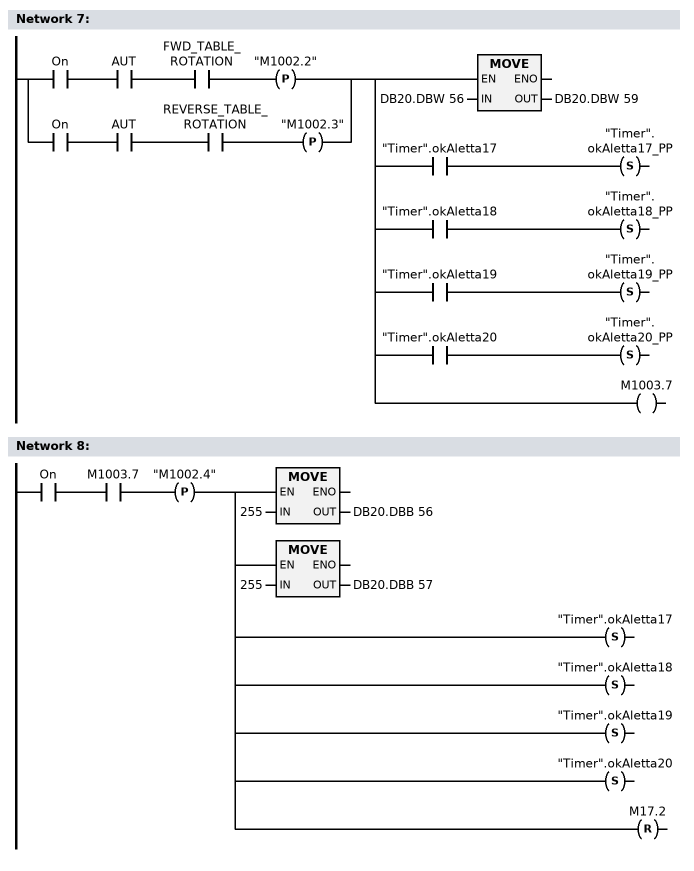
[picture p85: FC53 - REWORK networks 7-8]
NETWORK
TITLE =
      A     "On";
      A     "AUT";
      A     "FWD_TABLE_ROTATION";
      FP    "M1002.2";
      O(;
      A     "On";
      A     "AUT";
      A     "REVERSE_TABLE_ROTATION";
      FP    "M1002.3";
      );
      =     L 0.0;
      A     L 0.0;
      JNB   _009;
      L     DB20.DBW 56;
      T     DB20.DBW 59;
_009: NOP   0;
      A     L 0.0;
      A     "Timer".okAletta17;
      S     "Timer".okAletta17_PP;
      A     L 0.0;
      A     "Timer".okAletta18;
      S     "Timer".okAletta18_PP;
      A     L 0.0;
      A     "Timer".okAletta19;
      S     "Timer".okAletta19_PP;
      A     L 0.0;
      A     "Timer".okAletta20;
      S     "Timer".okAletta20_PP;
      A     L 0.0;
      BLD   102;
      =     "M1003.7";
NETWORK
TITLE =
      A     "On";
      A     "M1003.7";
      FP    "M1002.4";
      =     L 0.0;
      A     L 0.0;
      JNB   _00a;
      L     255;
      T     DB20.DBB 56;
_00a: NOP   0;
      A     L 0.0;
      JNB   _00b;
      L     255;
      T     DB20.DBB 57;
_00b: NOP   0;
      A     L 0.0;
      BLD   102;
      S     "Timer".okAletta17;
      A     L 0.0;
      BLD   102;
      S     "Timer".okAletta18;
      A     L 0.0;
      BLD   102;
      S     "Timer".okAletta19;
      A     L 0.0;
      BLD   102;
      S     "Timer".okAletta20;
      A     L 0.0;
      BLD   102;
      R     "M17.2";
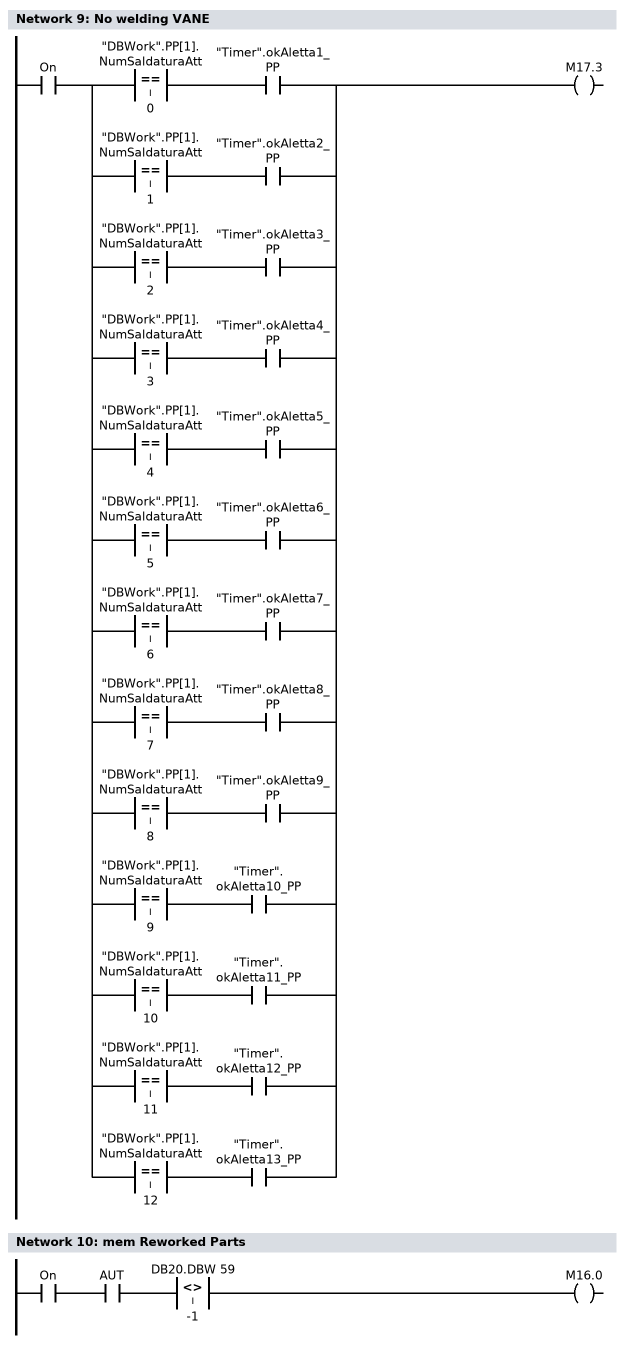
NETWORK
TITLE = No welding VANE
      A     "On";
      A(;
      A(;
      L     "DBWork".PP[1].NumSaldaturaAtt;
      L     0;
      ==I;
      );
      A     "Timer".okAletta1_PP;
      O;
      A(;
      L     "DBWork".PP[1].NumSaldaturaAtt;
      L     1;
      ==I;
      );
      A     "Timer".okAletta2_PP;
      O;
      A(;
      L     "DBWork".PP[1].NumSaldaturaAtt;
      L     2;
      ==I;
      );
      A     "Timer".okAletta3_PP;
      O;
      A(;
      L     "DBWork".PP[1].NumSaldaturaAtt;
      L     3;
      ==I;
      );
      A     "Timer".okAletta4_PP;
      O;
      A(;
      L     "DBWork".PP[1].NumSaldaturaAtt;
      L     4;
      ==I;
      );
      A     "Timer".okAletta5_PP;
      O;
      A(;
      L     "DBWork".PP[1].NumSaldaturaAtt;
      L     5;
      ==I;
      );
      A     "Timer".okAletta6_PP;
      O;
      A(;
      L     "DBWork".PP[1].NumSaldaturaAtt;
      L     6;
      ==I;
      );
      A     "Timer".okAletta7_PP;
      O;
      A(;
      L     "DBWork".PP[1].NumSaldaturaAtt;
      L     7;
      ==I;
      );
      A     "Timer".okAletta8_PP;
      O;
      A(;
      L     "DBWork".PP[1].NumSaldaturaAtt;
      L     8;
      ==I;
      );
      A     "Timer".okAletta9_PP;
      O;
      A(;
      L     "DBWork".PP[1].NumSaldaturaAtt;
      L     9;
      ==I;
      );
      A     "Timer".okAletta10_PP;
      O;
      A(;
      L     "DBWork".PP[1].NumSaldaturaAtt;
      L     10;
      ==I;
      );
      A     "Timer".okAletta11_PP;
      O;
      A(;
      L     "DBWork".PP[1].NumSaldaturaAtt;
      L     11;
      ==I;
      );
      A     "Timer".okAletta12_PP;
      O;
      A(;
      L     "DBWork".PP[1].NumSaldaturaAtt;
      L     12;
      ==I;
      );
      A     "Timer".okAletta13_PP;
      );
      =     "M17.3";
NETWORK
TITLE = mem Reworked Parts
      A     "On";
      A     "AUT";
      A(;
      L     DB20.DBW 59;
      L     -1;
      <>I;
      );
      =     "M16.0";
END_FUNCTION

FUNCTION "FC81 - GEST AXIS" : VOID	// FC 81
VERSION : 0.1
VAR_TEMP
  AttualPos : DINT ;
  AttualPosR : REAL ;
  Override : INT ;
  AuxRelative : DINT ;
  JogRelative : BOOL ;
END_VAR
BEGIN
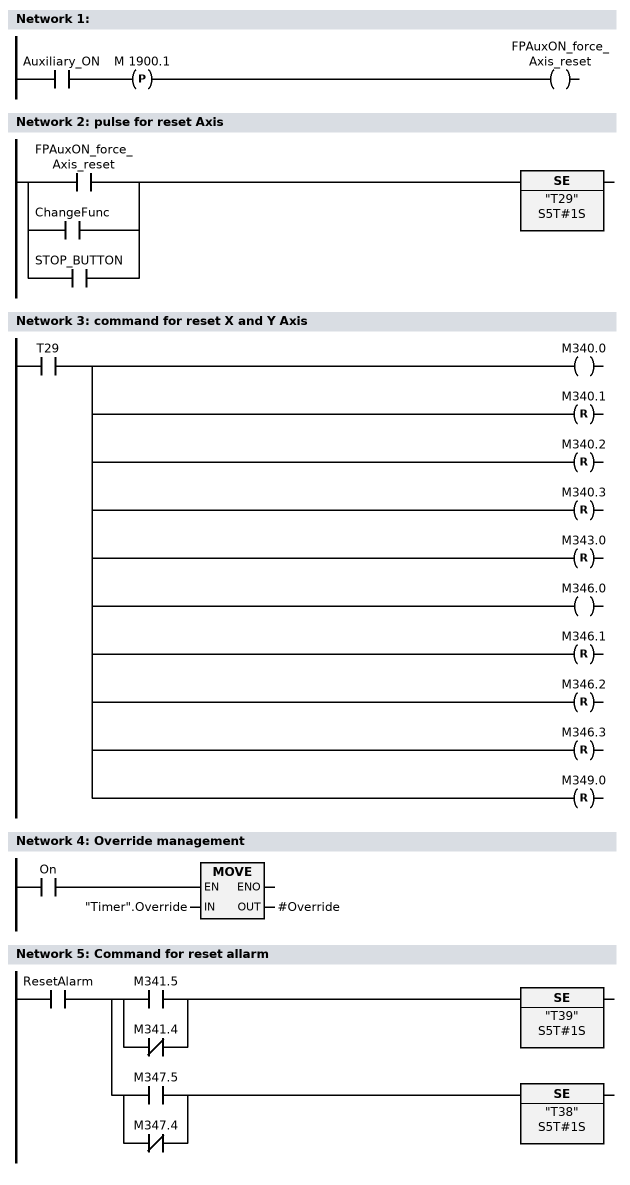
NETWORK
TITLE =
      A     "Auxiliary_ON";
      FP    M 1900.1;
      =     "FPAuxON_force_Axis_reset";
NETWORK
TITLE = pulse for reset Axis
      O     "FPAuxON_force_Axis_reset";
      O     "ChangeFunc";
      O     "STOP_BUTTON";
      L     S5T#1S;
      SE    "T29";
NETWORK
TITLE = command for reset X and Y Axis
      A     "T29";
      =     "M340.0";
      R     "M340.1";
      R     "M340.2";
      R     "M340.3";
      R     "M343.0";
      =     "M346.0";
      R     "M346.1";
      R     "M346.2";
      R     "M346.3";
      R     "M349.0";
NETWORK
TITLE = Override management
//"DatiMacchina".AcesXYZC_Override_Aux
      A     "On";
      JNB   _001;
      L     "Timer".Override;
      T     #Override;
_001: NOP   0;
NETWORK
TITLE = Command for reset allarm
      A     "ResetAlarm";
      =     L 15.0;
      A     L 15.0;
      A(;
      O     "M341.5";
      ON    "M341.4";
      );
      L     S5T#1S;
      SE    "T39";
      A     L 15.0;
      A(;
      O     "M347.5";
      ON    "M347.4";
      );
      L     S5T#1S;
      SE    "T38";
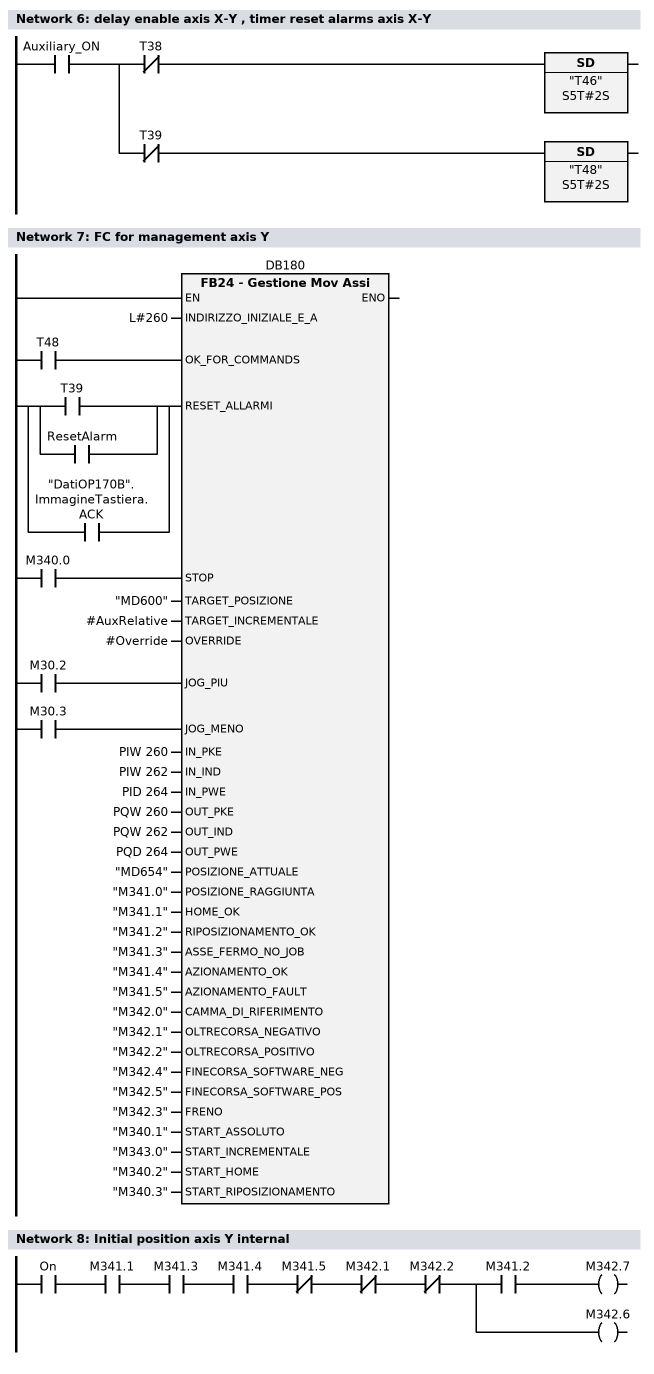
NETWORK
TITLE = delay enable axis X-Y , timer reset alarms axis X-Y
      A     "Auxiliary_ON";
      =     L 15.0;
      A     L 15.0;
      AN    "T38";
      L     S5T#2S;
      SD    "T46";
      A     L 15.0;
      AN    "T39";
      L     S5T#2S;
      SD    "T48";
NETWORK
TITLE = FC for management axis Y
      A     "T48";
      =     L 15.0;
      BLD   103;
      A(;
      O     "T39";
      O     "ResetAlarm";
      O     "DatiOP170B".ImmagineTastiera.ACK;
      );
      =     L 15.1;
      BLD   103;
      A     "M340.0";
      =     L 15.2;
      BLD   103;
      A     "M30.2";
      =     L 15.3;
      BLD   103;
      A     "M30.3";
      =     L 15.4;
      BLD   103;
      CALL  "FB24 - Gestione Mov Assi" , "DB180" (
           INDIRIZZO_INIZIALE_E_A   := L#260,
           OK_FOR_COMMANDS          := L 15.0,
           RESET_ALLARMI            := L 15.1,
           STOP                     := L 15.2,
           TARGET_POSIZIONE         := "MD600",
           TARGET_INCREMENTALE      := #AuxRelative,
           OVERRIDE                 := #Override,
           JOG_PIU                  := L 15.3,
           JOG_MENO                 := L 15.4,
           IN_PKE                   := PIW 260,
           IN_IND                   := PIW 262,
           IN_PWE                   := PID 264,
           OUT_PKE                  := PQW 260,
           OUT_IND                  := PQW 262,
           OUT_PWE                  := PQD 264,
           POSIZIONE_ATTUALE        := "MD654",
           POSIZIONE_RAGGIUNTA      := "M341.0",
           HOME_OK                  := "M341.1",
           RIPOSIZIONAMENTO_OK      := "M341.2",
           ASSE_FERMO_NO_JOB        := "M341.3",
           AZIONAMENTO_OK           := "M341.4",
           AZIONAMENTO_FAULT        := "M341.5",
           CAMMA_DI_RIFERIMENTO     := "M342.0",
           OLTRECORSA_NEGATIVO      := "M342.1",
           OLTRECORSA_POSITIVO      := "M342.2",
           FINECORSA_SOFTWARE_NEG   := "M342.4",
           FINECORSA_SOFTWARE_POS   := "M342.5",
           FRENO                    := "M342.3",
           START_ASSOLUTO           := "M340.1",
           START_INCREMENTALE       := "M343.0",
           START_HOME               := "M340.2",
           START_RIPOSIZIONAMENTO   := "M340.3");
      NOP   0;
NETWORK
TITLE = Initial position axis Y internal
      A     "On";
      A     "M341.1";
      A     "M341.3";
      A     "M341.4";
      AN    "M341.5";
      AN    "M342.1";
      AN    "M342.2";
      =     L 15.0;
      A     L 15.0;
      A     "M341.2";
      =     "M342.7";
      A     L 15.0;
      BLD   102;
      =     "M342.6";
NETWORK
TITLE = Axis X Management
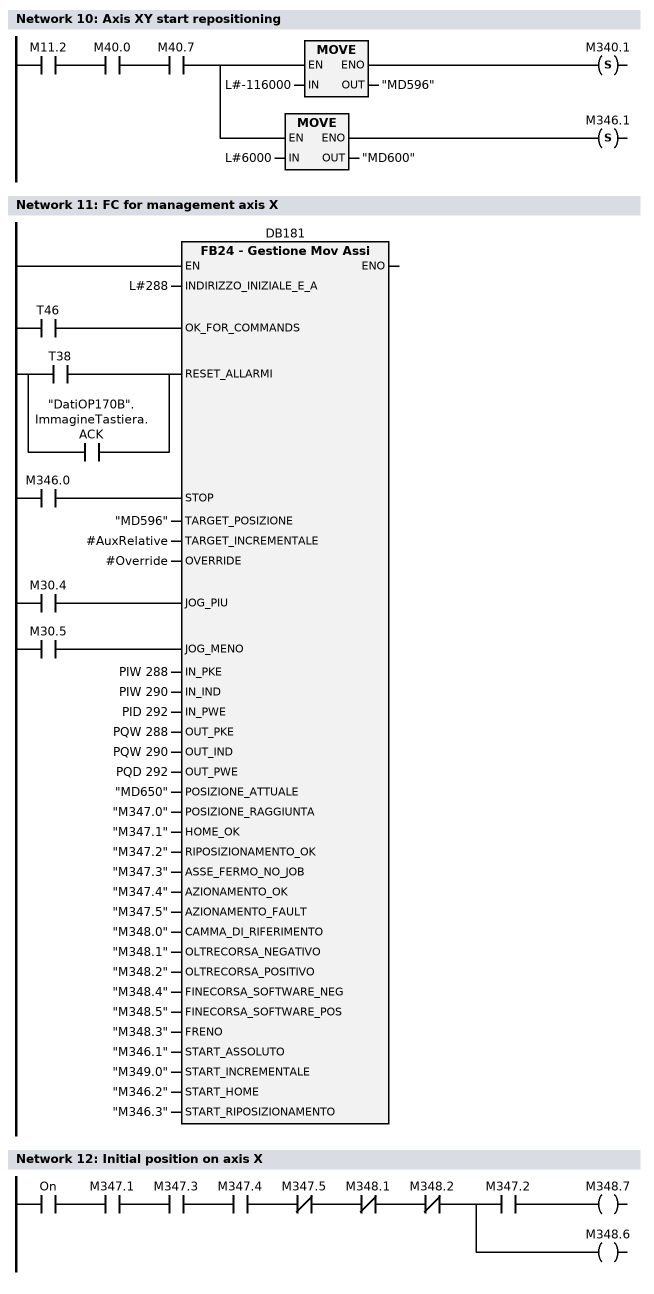
NETWORK
TITLE = Axis XY start repositioning
      A     "M11.2";
      A     "M40.0";
      A     "M40.7";
      =     L 15.0;
      A     L 15.0;
      JNB   _002;
      L     L#-116000;
      T     "MD596";
      SET;
      SAVE;
      CLR;
_002: A     BR;
      S     "M340.1";
      A     L 15.0;
      JNB   _003;
      L     L#6000;
      T     "MD600";
      SET;
      SAVE;
      CLR;
_003: A     BR;
      S     "M346.1";
NETWORK
TITLE = FC for management axis X
      A     "T46";
      =     L 15.0;
      BLD   103;
      A(;
      O     "T38";
      O     "DatiOP170B".ImmagineTastiera.ACK;
      );
      =     L 15.1;
      BLD   103;
      A     "M346.0";
      =     L 15.2;
      BLD   103;
      A     "M30.4";
      =     L 15.3;
      BLD   103;
      A     "M30.5";
      =     L 15.4;
      BLD   103;
      CALL  "FB24 - Gestione Mov Assi" , "DB181" (
           INDIRIZZO_INIZIALE_E_A   := L#288,
           OK_FOR_COMMANDS          := L 15.0,
           RESET_ALLARMI            := L 15.1,
           STOP                     := L 15.2,
           TARGET_POSIZIONE         := "MD596",
           TARGET_INCREMENTALE      := #AuxRelative,
           OVERRIDE                 := #Override,
           JOG_PIU                  := L 15.3,
           JOG_MENO                 := L 15.4,
           IN_PKE                   := PIW 288,
           IN_IND                   := PIW 290,
           IN_PWE                   := PID 292,
           OUT_PKE                  := PQW 288,
           OUT_IND                  := PQW 290,
           OUT_PWE                  := PQD 292,
           POSIZIONE_ATTUALE        := "MD650",
           POSIZIONE_RAGGIUNTA      := "M347.0",
           HOME_OK                  := "M347.1",
           RIPOSIZIONAMENTO_OK      := "M347.2",
           ASSE_FERMO_NO_JOB        := "M347.3",
           AZIONAMENTO_OK           := "M347.4",
           AZIONAMENTO_FAULT        := "M347.5",
           CAMMA_DI_RIFERIMENTO     := "M348.0",
           OLTRECORSA_NEGATIVO      := "M348.1",
           OLTRECORSA_POSITIVO      := "M348.2",
           FINECORSA_SOFTWARE_NEG   := "M348.4",
           FINECORSA_SOFTWARE_POS   := "M348.5",
           FRENO                    := "M348.3",
           START_ASSOLUTO           := "M346.1",
           START_INCREMENTALE       := "M349.0",
           START_HOME               := "M346.2",
           START_RIPOSIZIONAMENTO   := "M346.3");
      NOP   0;
NETWORK
TITLE = Initial position on axis X
      A     "On";
      A     "M347.1";
      A     "M347.3";
      A     "M347.4";
      AN    "M347.5";
      AN    "M348.1";
      AN    "M348.2";
      =     L 15.0;
      A     L 15.0;
      A     "M347.2";
      =     "M348.7";
      A     L 15.0;
      BLD   102;
      =     "M348.6";
END_FUNCTION

FUNCTION "FC117 - ERROR TOOL" : VOID	// FC 117
VERSION : 0.1
BEGIN
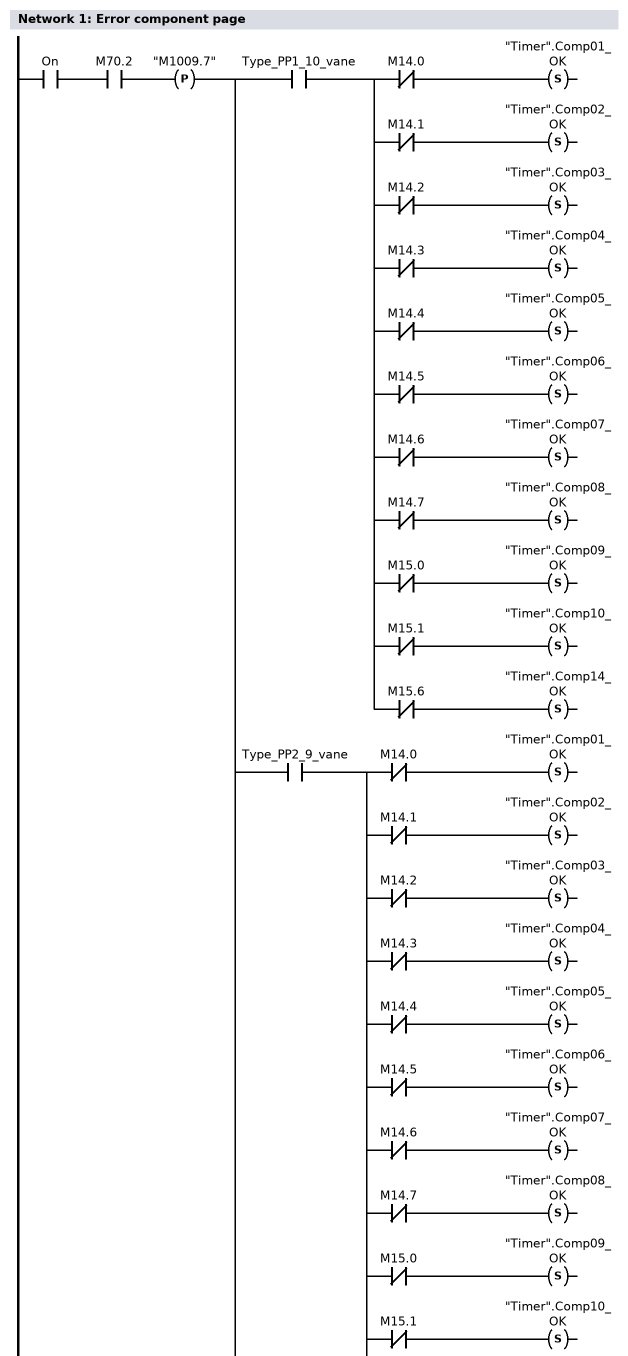
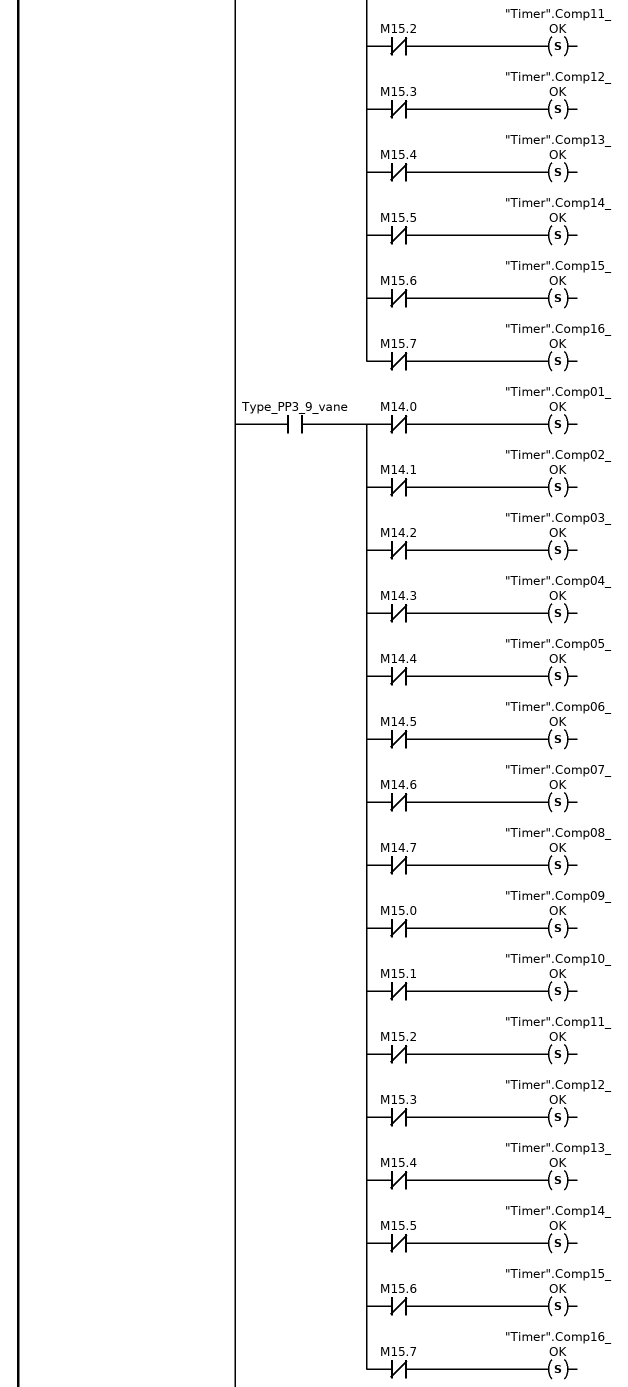
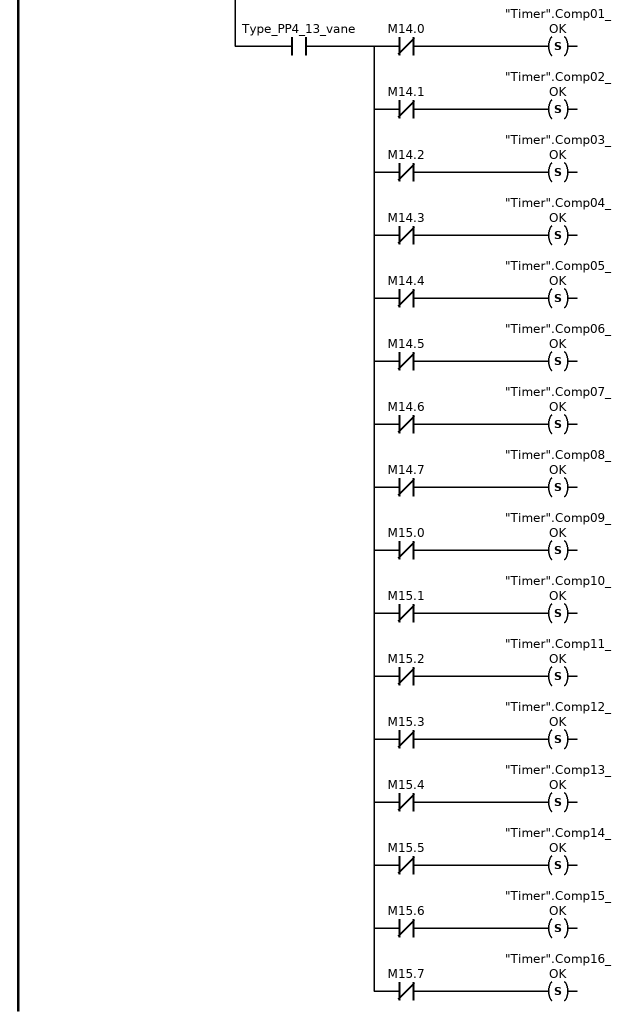
NETWORK
TITLE = Error component page
      A     "On";
      A     "M70.2";
      FP    "M1009.7";
      =     L 0.0;
      A     L 0.0;
      A     "Type_PP1_10_vane";
      =     L 0.1;
      A     L 0.1;
      AN    "M14.0";
      S     "Timer".Comp01_OK;
      A     L 0.1;
      AN    "M14.1";
      S     "Timer".Comp02_OK;
      A     L 0.1;
      AN    "M14.2";
      S     "Timer".Comp03_OK;
      A     L 0.1;
      AN    "M14.3";
      S     "Timer".Comp04_OK;
      A     L 0.1;
      AN    "M14.4";
      S     "Timer".Comp05_OK;
      A     L 0.1;
      AN    "M14.5";
      S     "Timer".Comp06_OK;
      A     L 0.1;
      AN    "M14.6";
      S     "Timer".Comp07_OK;
      A     L 0.1;
      AN    "M14.7";
      S     "Timer".Comp08_OK;
      A     L 0.1;
      AN    "M15.0";
      S     "Timer".Comp09_OK;
      A     L 0.1;
      AN    "M15.1";
      S     "Timer".Comp10_OK;
      A     L 0.1;
      AN    "M15.6";
      S     "Timer".Comp14_OK;
      A     L 0.0;
      A     "Type_PP2_9_vane";
      =     L 0.1;
      A     L 0.1;
      AN    "M14.0";
      S     "Timer".Comp01_OK;
      A     L 0.1;
      AN    "M14.1";
      S     "Timer".Comp02_OK;
      A     L 0.1;
      AN    "M14.2";
      S     "Timer".Comp03_OK;
      A     L 0.1;
      AN    "M14.3";
      S     "Timer".Comp04_OK;
      A     L 0.1;
      AN    "M14.4";
      S     "Timer".Comp05_OK;
      A     L 0.1;
      AN    "M14.5";
      S     "Timer".Comp06_OK;
      A     L 0.1;
      AN    "M14.6";
      S     "Timer".Comp07_OK;
      A     L 0.1;
      AN    "M14.7";
      S     "Timer".Comp08_OK;
      A     L 0.1;
      AN    "M15.0";
      S     "Timer".Comp09_OK;
      A     L 0.1;
      AN    "M15.1";
      S     "Timer".Comp10_OK;
      A     L 0.1;
      AN    "M15.2";
      S     "Timer".Comp11_OK;
      A     L 0.1;
      AN    "M15.3";
      S     "Timer".Comp12_OK;
      A     L 0.1;
      AN    "M15.4";
      S     "Timer".Comp13_OK;
      A     L 0.1;
      AN    "M15.5";
      S     "Timer".Comp14_OK;
      A     L 0.1;
      AN    "M15.6";
      S     "Timer".Comp15_OK;
      A     L 0.1;
      AN    "M15.7";
      S     "Timer".Comp16_OK;
      A     L 0.0;
      A     "Type_PP3_9_vane";
      =     L 0.1;
      A     L 0.1;
      AN    "M14.0";
      S     "Timer".Comp01_OK;
      A     L 0.1;
      AN    "M14.1";
      S     "Timer".Comp02_OK;
      A     L 0.1;
      AN    "M14.2";
      S     "Timer".Comp03_OK;
      A     L 0.1;
      AN    "M14.3";
      S     "Timer".Comp04_OK;
      A     L 0.1;
      AN    "M14.4";
      S     "Timer".Comp05_OK;
      A     L 0.1;
      AN    "M14.5";
      S     "Timer".Comp06_OK;
      A     L 0.1;
      AN    "M14.6";
      S     "Timer".Comp07_OK;
      A     L 0.1;
      AN    "M14.7";
      S     "Timer".Comp08_OK;
      A     L 0.1;
      AN    "M15.0";
      S     "Timer".Comp09_OK;
      A     L 0.1;
      AN    "M15.1";
      S     "Timer".Comp10_OK;
      A     L 0.1;
      AN    "M15.2";
      S     "Timer".Comp11_OK;
      A     L 0.1;
      AN    "M15.3";
      S     "Timer".Comp12_OK;
      A     L 0.1;
      AN    "M15.4";
      S     "Timer".Comp13_OK;
      A     L 0.1;
      AN    "M15.5";
      S     "Timer".Comp14_OK;
      A     L 0.1;
      AN    "M15.6";
      S     "Timer".Comp15_OK;
      A     L 0.1;
      AN    "M15.7";
      S     "Timer".Comp16_OK;
      A     L 0.0;
      A     "Type_PP4_13_vane";
      =     L 0.1;
      A     L 0.1;
      AN    "M14.0";
      S     "Timer".Comp01_OK;
      A     L 0.1;
      AN    "M14.1";
      S     "Timer".Comp02_OK;
      A     L 0.1;
      AN    "M14.2";
      S     "Timer".Comp03_OK;
      A     L 0.1;
      AN    "M14.3";
      S     "Timer".Comp04_OK;
      A     L 0.1;
      AN    "M14.4";
      S     "Timer".Comp05_OK;
      A     L 0.1;
      AN    "M14.5";
      S     "Timer".Comp06_OK;
      A     L 0.1;
      AN    "M14.6";
      S     "Timer".Comp07_OK;
      A     L 0.1;
      AN    "M14.7";
      S     "Timer".Comp08_OK;
      A     L 0.1;
      AN    "M15.0";
      S     "Timer".Comp09_OK;
      A     L 0.1;
      AN    "M15.1";
      S     "Timer".Comp10_OK;
      A     L 0.1;
      AN    "M15.2";
      S     "Timer".Comp11_OK;
      A     L 0.1;
      AN    "M15.3";
      S     "Timer".Comp12_OK;
      A     L 0.1;
      AN    "M15.4";
      S     "Timer".Comp13_OK;
      A     L 0.1;
      AN    "M15.5";
      S     "Timer".Comp14_OK;
      A     L 0.1;
      AN    "M15.6";
      S     "Timer".Comp15_OK;
      A     L 0.1;
      AN    "M15.7";
      S     "Timer".Comp16_OK;
END_FUNCTION

FUNCTION "TimeOut" : VOID	// FC 800
TITLE = Gestione timeout movimento
FAMILY : GCLib
NAME : TimeOut
VERSION : 1.0
VAR_INPUT
  Condizione1 : BOOL ;
  Condizione2 : BOOL ;
  Contatore : COUNTER ;
  Reset : BOOL ;
  Tempo_TimeOut : INT ;
END_VAR
VAR_IN_OUT
  TimeOut_Condizione1 : BOOL ;
  TimeOut_Condizione2 : BOOL ;
END_VAR
BEGIN
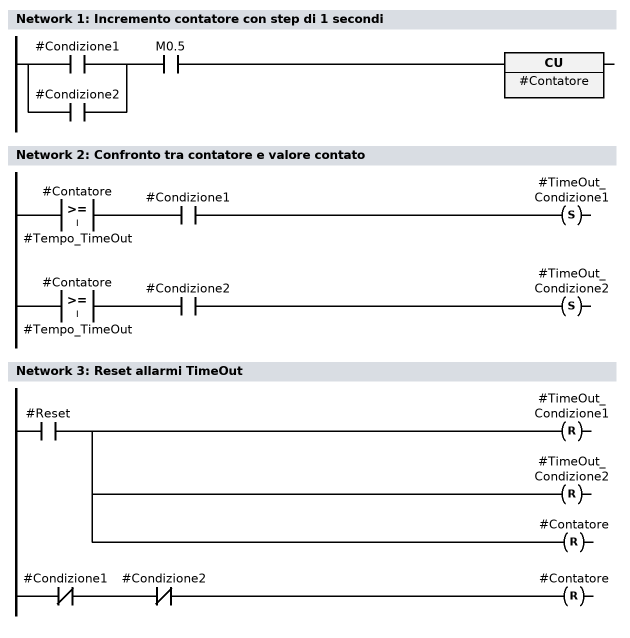
NETWORK
TITLE = Incremento contatore con step di 1 secondi
      A     #Condizione1;
      O     #Condizione2;
      A     "M0.5";
      CU    #Contatore;
NETWORK
TITLE = Confronto tra contatore e valore contato
      L     #Contatore;
      L     #Tempo_TimeOut;
      >=I;
      A     #Condizione1;
      S     #TimeOut_Condizione1;
      L     #Contatore;
      L     #Tempo_TimeOut;
      >=I;
      A     #Condizione2;
      S     #TimeOut_Condizione2;
NETWORK
TITLE = Reset allarmi TimeOut
      A     #Reset;
      R     #TimeOut_Condizione1;
      R     #TimeOut_Condizione2;
      R     #Contatore;
      AN    #Condizione1;
      AN    #Condizione2;
      R     #Contatore;
END_FUNCTION

DATA_BLOCK "DI_Balluff1"	// DB 5
VERSION : 0.0
"BALLUFF"
BEGIN
END_DATA_BLOCK

DATA_BLOCK "DatiOP170B"	// DB 7
TITLE = Dati interfaccia tra PLC e OP170B
FAMILY : GCLib
VERSION : 0.1
  STRUCT
   NumeroPagina : STRUCT
    TipoPaginaCorrente : WORD ;
    NumeroPaginaCorrente : INT ;
    Riservato1 : WORD ;
    Riservato2 : WORD ;
    Riservato3 : WORD ;
   END_STRUCT ;
   BufferOrdini : STRUCT
    NU : BYTE ;
    NumeroOrdine : BYTE ;
    Parametro1 : WORD ;
    Parametro2 : WORD ;
    Parametro3 : WORD ;
   END_STRUCT ;
   Coordinazione : STRUCT
    NU : BYTE ;
    BitAvvio : BOOL ;
    TipoFunzionamento : BOOL ;
    BitAttivita : BOOL ;
    Riservato1 : BOOL ;
    Riservato2 : BOOL ;
    Riservato3 : BOOL ;
    Riservato4 : BOOL ;
    Riservato5 : BOOL ;
    Riservata : WORD ;
   END_STRUCT ;
   ImmagineLED : STRUCT
    Bit0_F1 : BOOL ;
    Bit1_F1 : BOOL ;
    Bit0_F2 : BOOL ;
    Bit1_F2 : BOOL ;
    Bit0_F3 : BOOL ;
    Bit1_F3 : BOOL ;
    Bit0_F4 : BOOL ;
    Bit1_F4 : BOOL ;
    Bit0_F5 : BOOL ;
    Bit1_F5 : BOOL ;
    Bit0_F6 : BOOL ;
    Bit1_F6 : BOOL ;
    Bit0_F7 : BOOL ;
    Bit1_F7 : BOOL ;
    Bit0_F8 : BOOL ;
    Bit1_F8 : BOOL ;
    Bit0_K1 : BOOL ;
    Bit1_K1 : BOOL ;
    Bit0_K2 : BOOL ;
    Bit1_K2 : BOOL ;
    Bit0_K3 : BOOL ;
    Bit1_K3 : BOOL ;
    Bit0_K4 : BOOL ;
    Bit1_K4 : BOOL ;
    Bit0_K5 : BOOL ;
    Bit1_K5 : BOOL ;
    Bit0_K6 : BOOL ;
    Bit1_K6 : BOOL ;
    Bit0_K7 : BOOL ;
    Bit1_K7 : BOOL ;
    Bit0_K8 : BOOL ;
    Bit1_K8 : BOOL ;
    Bit0_K9 : BOOL ;
    Bit1_K9 : BOOL ;
    Bit0_K10 : BOOL ;
    Bit1_K10 : BOOL ;
    NU1 : BOOL ;
    NU2 : BOOL ;
    NU3 : BOOL ;
    NU4 : BOOL ;
    NU5 : BOOL ;
    NU6 : BOOL ;
    NU7 : BOOL ;
    NU8 : BOOL ;
    NU9 : BOOL ;
    NU10 : BOOL ;
    NU11 : BOOL ;
    NU12 : BOOL ;
   END_STRUCT ;
   ImmagineTastiera : STRUCT
    F1 : BOOL ;
    F2 : BOOL ;
    F3 : BOOL ;
    F4 : BOOL ;
    F5 : BOOL ;
    F6 : BOOL ;
    F7 : BOOL ;
    F8 : BOOL ;
    F9 : BOOL ;
    F10 : BOOL ;
    F11 : BOOL ;
    F12 : BOOL ;
    F13 : BOOL ;
    F14 : BOOL ;
    K1 : BOOL ;
    K2 : BOOL ;
    K3 : BOOL ;
    K4 : BOOL ;
    K5 : BOOL ;
    K6 : BOOL ;
    K7 : BOOL ;
    K8 : BOOL ;
    K9 : BOOL ;
    K10 : BOOL ;
    DEC_1_K13 : BOOL ;
    INC_1_K12 : BOOL ;
    HELP : BOOL ;
    ESC : BOOL ;
    ACK : BOOL ;
    ENTER : BOOL ;
    NU7 : BOOL ;
    NU8 : BOOL ;
   END_STRUCT ;
   PLCDataOra : DATE_AND_TIME ;
   PLCDataOraNU : DWORD ;
   SegnalazioniServizio : STRUCT
    TEXT9 : BOOL ;
    TEXT10 : BOOL ;
    TEXT11 : BOOL ;
    TEXT12 : BOOL ;
    TEXT13 : BOOL ;
    TEXT14 : BOOL ;
    TEXT15 : BOOL ;
    TEXT16 : BOOL ;
    TEXT1 : BOOL ;
    TEXT2 : BOOL ;
    TEXT3 : BOOL ;
    TEXT4 : BOOL ;
    TEXT5 : BOOL ;
    TEXT6 : BOOL ;
    TEXT7 : BOOL ;
    TEXT8 : BOOL ;
    TEXT25 : BOOL ;
    TEXT26 : BOOL ;
    TEXT27 : BOOL ;
    TEXT28 : BOOL ;
    TEXT29 : BOOL ;
    TEXT30 : BOOL ;
    TEXT31 : BOOL ;
    TEXT32 : BOOL ;
    TEXT17 : BOOL ;
    TEXT18 : BOOL ;
    TEXT19 : BOOL ;
    TEXT20 : BOOL ;
    TEXT21 : BOOL ;
    TEXT22 : BOOL ;
    TEXT23 : BOOL ;
    TEXT24 : BOOL ;
    TEXT41 : BOOL ;
    TEXT42 : BOOL ;
    TEXT43 : BOOL ;
    TEXT44 : BOOL ;
    TEXT45 : BOOL ;
    TEXT46 : BOOL ;
    TEXT47 : BOOL ;
    TEXT48 : BOOL ;
    TEXT33 : BOOL ;
    TEXT34 : BOOL ;
    TEXT35 : BOOL ;
    TEXT36 : BOOL ;
    TEXT37 : BOOL ;
    TEXT38 : BOOL ;
    TEXT39 : BOOL ;
    TEXT40 : BOOL ;
    TEXT57 : BOOL ;
    TEXT58 : BOOL ;
    TEXT59 : BOOL ;
    TEXT60 : BOOL ;
    TEXT61 : BOOL ;
    TEXT62 : BOOL ;
    TEXT63 : BOOL ;
    TEXT64 : BOOL ;
    TEXT49 : BOOL ;
    TEXT50 : BOOL ;
    TEXT51 : BOOL ;
    TEXT52 : BOOL ;
    TEXT53 : BOOL ;
    TEXT54 : BOOL ;
    TEXT55 : BOOL ;
    TEXT56 : BOOL ;
    TEXT73 : BOOL ;
    TEXT74 : BOOL ;
    TEXT75 : BOOL ;
    TEXT76 : BOOL ;
    TEXT77 : BOOL ;
    TEXT78 : BOOL ;
    TEXT79 : BOOL ;
    TEXT80 : BOOL ;
    TEXT65 : BOOL ;
    TEXT66 : BOOL ;
    TEXT67 : BOOL ;
    TEXT68 : BOOL ;
    TEXT69 : BOOL ;
    TEXT70 : BOOL ;
    TEXT71 : BOOL ;
    TEXT72 : BOOL ;
    TEXT89 : BOOL ;
    TEXT90 : BOOL ;
    TEXT91 : BOOL ;
    TEXT92 : BOOL ;
    TEXT93 : BOOL ;
    TEXT94 : BOOL ;
    TEXT95 : BOOL ;
    TEXT96 : BOOL ;	//TEXT N.96
    TEXT81 : BOOL ;
    TEXT82 : BOOL ;	//TEXT N.82
    TEXT83 : BOOL ;	//TEXT N.83
    TEXT84 : BOOL ;	//TEXT N.84
    TEXT85 : BOOL ;	//TEXT N.85
    TEXT86 : BOOL ;	//TEXT N.86
    TEXT87 : BOOL ;	//TEXT N.87
    TEXT88 : BOOL ;	//TEXT N.88
    TEXT105 : BOOL ;	//TEXT N.105
    TEXT106 : BOOL ;	//TEXT N.106
    TEXT107 : BOOL ;	//TEXT N.107
    TEXT108 : BOOL ;	//TEXT N.108
    TEXT109 : BOOL ;	//TEXT N.109
    TEXT110 : BOOL ;	//TEXT N.110
    TEXT111 : BOOL ;	//TEXT N.111
    TEXT112 : BOOL ;	//TEXT N.112
    TEXT97 : BOOL ;	//TEXT N.17
    TEXT98 : BOOL ;	//TEXT N.18
    TEXT99 : BOOL ;	//TEXT N.19
    TEXT100 : BOOL ;	//TEXT N.100
    TEXT101 : BOOL ;	//TEXT N.101
    TEXT102 : BOOL ;	//TEXT N.102
    TEXT103 : BOOL ;	//TEXT N.103
    TEXT104 : BOOL ;	//TEXT N.104
    TEXT121 : BOOL ;	//TEXT N.121
    TEXT122 : BOOL ;	//TEXT N.122
    TEXT123 : BOOL ;	//TEXT N.123
    TEXT124 : BOOL ;	//TEXT N.124
    TEXT125 : BOOL ;	//TEXT N.125
    TEXT126 : BOOL ;	//TEXT N.126
    TEXT127 : BOOL ;	//TEXT N.127
    TEXT128 : BOOL ;	//TEXT N.128
    TEXT113 : BOOL ;	//TEXT N.113
    TEXT114 : BOOL ;	//TEXT N.114
    TEXT115 : BOOL ;	//TEXT N.115
    TEXT116 : BOOL ;	//TEXT N.116
    TEXT117 : BOOL ;	//TEXT N.117
    TEXT118 : BOOL ;	//TEXT N.118
    TEXT119 : BOOL ;	//TEXT N.119
    TEXT120 : BOOL ;	//TEXT N.120
    TEXT137 : BOOL ;	//TEXT N.137
    TEXT138 : BOOL ;	//TEXT N.138
    TEXT139 : BOOL ;	//TEXT N.139
    TEXT140 : BOOL ;	//TEXT N.140
    TEXT141 : BOOL ;	//TEXT N.141
    TEXT142 : BOOL ;	//TEXT N.142
    TEXT143 : BOOL ;	//TEXT N.143
    TEXT144 : BOOL ;	//TEXT N.144
    TEXT129 : BOOL ;	//TEXT N.129
    TEXT130 : BOOL ;	//TEXT N.130
    TEXT131 : BOOL ;	//TEXT N.131
    TEXT132 : BOOL ;	//TEXT N.132
    TEXT133 : BOOL ;	//TEXT N.133
    TEXT134 : BOOL ;	//TEXT N.134
    TEXT135 : BOOL ;	//TEXT N.135
    TEXT136 : BOOL ;	//TEXT N.136
    TEXT153 : BOOL ;	//TEXT N.153
    TEXT154 : BOOL ;	//TEXT N.154
    TEXT155 : BOOL ;	//TEXT N.155
    TEXT156 : BOOL ;	//TEXT N.156
    TEXT157 : BOOL ;	//TEXT N.157
    TEXT158 : BOOL ;	//TEXT N.158
    TEXT159 : BOOL ;	//TEXT N.159
    TEXT160 : BOOL ;	//TEXT N.160
    TEXT145 : BOOL ;	//TEXT N.145
    TEXT146 : BOOL ;	//TEXT N.146
    TEXT147 : BOOL ;	//TEXT N.147
    TEXT148 : BOOL ;	//TEXT N.148
    TEXT149 : BOOL ;	//TEXT N.149
    TEXT150 : BOOL ;	//TEXT N.150
    TEXT151 : BOOL ;	//TEXT N.151
    TEXT152 : BOOL ;	//TEXT N.152
    TEXT169 : BOOL ;	//TEXT N.169
    TEXT170 : BOOL ;	//TEXT N.170
    TEXT171 : BOOL ;	//TEXT N.171
    TEXT172 : BOOL ;	//TEXT N.172
    TEXT173 : BOOL ;	//TEXT N.173
    TEXT174 : BOOL ;	//TEXT N.174
    TEXT175 : BOOL ;	//TEXT N.175
    TEXT176 : BOOL ;	//TEXT N.176
    TEXT161 : BOOL ;	//TEXT N.161
    TEXT162 : BOOL ;	//TEXT N.162
    TEXT163 : BOOL ;	//TEXT N.163
    TEXT164 : BOOL ;	//TEXT N.164
    TEXT165 : BOOL ;	//TEXT N.165
    TEXT166 : BOOL ;	//TEXT N.166
    TEXT167 : BOOL ;	//TEXT N.167
    TEXT168 : BOOL ;	//TEXT N.168
    TEXT185 : BOOL ;	//TEXT N.185
    TEXT186 : BOOL ;	//TEXT N.186
    TEXT187 : BOOL ;	//TEXT N.187
    TEXT188 : BOOL ;	//TEXT N.188
    TEXT189 : BOOL ;	//TEXT N.189
    TEXT190 : BOOL ;	//TEXT N.190
    TEXT191 : BOOL ;	//TEXT N.191
    TEXT192 : BOOL ;	//TEXT N.192
    TEXT177 : BOOL ;	//TEXT N.177
    TEXT178 : BOOL ;	//TEXT N.178
    TEXT179 : BOOL ;	//TEXT N.179
    TEXT180 : BOOL ;	//TEXT N.180
    TEXT181 : BOOL ;	//TEXT N.181
    TEXT182 : BOOL ;	//TEXT N.182
    TEXT183 : BOOL ;	//TEXT N.183
    TEXT184 : BOOL ;	//TEXT N.184
    TEXT201 : BOOL ;	//TEXT N.201
    TEXT202 : BOOL ;	//TEXT N.202
    TEXT203 : BOOL ;	//TEXT N.203
    TEXT204 : BOOL ;	//TEXT N.204
    TEXT205 : BOOL ;	//TEXT N.205
    TEXT206 : BOOL ;	//TEXT N.206
    TEXT207 : BOOL ;	//TEXT N.207
    TEXT208 : BOOL ;	//TEXT N.208
    TEXT193 : BOOL ;	//TEXT N.193
    TEXT194 : BOOL ;	//TEXT N.194
    TEXT195 : BOOL ;	//TEXT N.195
    TEXT196 : BOOL ;	//TEXT N.196
    TEXT197 : BOOL ;	//TEXT N.197
    TEXT198 : BOOL ;	//TEXT N.198
    TEXT199 : BOOL ;	//TEXT N.199
    TEXT200 : BOOL ;	//TEXT N.200
    TEXT217 : BOOL ;	//TEXT N.217
    TEXT218 : BOOL ;	//TEXT N.218
    TEXT219 : BOOL ;	//TEXT N.219
    TEXT220 : BOOL ;	//TEXT N.220
    TEXT221 : BOOL ;	//TEXT N.221
    TEXT222 : BOOL ;	//TEXT N.222
    TEXT223 : BOOL ;	//TEXT N.223
    TEXT224 : BOOL ;	//TEXT N.224
    TEXT209 : BOOL ;	//TEXT N.209
    TEXT210 : BOOL ;	//TEXT N.210
    TEXT211 : BOOL ;	//TEXT N.211
    TEXT212 : BOOL ;	//TEXT N.212
    TEXT213 : BOOL ;	//TEXT N.213
    TEXT214 : BOOL ;	//TEXT N.214
    TEXT215 : BOOL ;	//TEXT N.215
    TEXT216 : BOOL ;	//TEXT N.216
    TEXT233 : BOOL ;	//TEXT N.233
    TEXT234 : BOOL ;	//TEXT N.234
    TEXT235 : BOOL ;	//TEXT N.235
    TEXT236 : BOOL ;	//TEXT N.236
    TEXT237 : BOOL ;	//TEXT N.237
    TEXT238 : BOOL ;	//TEXT N.238
    TEXT239 : BOOL ;	//TEXT N.239
    TEXT240 : BOOL ;	//TEXT N.240
    TEXT225 : BOOL ;	//TEXT N.225
    TEXT226 : BOOL ;	//TEXT N.226
    TEXT227 : BOOL ;	//TEXT N.227
    TEXT228 : BOOL ;	//TEXT N.228
    TEXT229 : BOOL ;	//TEXT N.229
    TEXT230 : BOOL ;	//TEXT N.230
    TEXT231 : BOOL ;	//TEXT N.231
    TEXT232 : BOOL ;	//TEXT N.232
    TEXT249 : BOOL ;	//TEXT N.249
    TEXT250 : BOOL ;	//TEXT N.250
    TEXT251 : BOOL ;	//TEXT N.251
    TEXT252 : BOOL ;	//TEXT N.252
    TEXT253 : BOOL ;	//TEXT N.253
    TEXT254 : BOOL ;	//TEXT N.254
    TEXT255 : BOOL ;	//TEXT N.255
    TEXT256 : BOOL ;	//TEXT N.256
    TEXT241 : BOOL ;	//TEXT N.241
    TEXT242 : BOOL ;	//TEXT N.242
    TEXT243 : BOOL ;	//TEXT N.243
    TEXT244 : BOOL ;	//TEXT N.244
    TEXT245 : BOOL ;	//TEXT N.245
    TEXT246 : BOOL ;	//TEXT N.246
    TEXT247 : BOOL ;	//TEXT N.247
    TEXT248 : BOOL ;	//TEXT N.248
    TEXT265 : BOOL ;	//TEXT N.265
    TEXT266 : BOOL ;	//TEXT N.266
    TEXT267 : BOOL ;	//TEXT N.267
    TEXT268 : BOOL ;	//TEXT N.268
    TEXT269 : BOOL ;	//TEXT N.269
    TEXT270 : BOOL ;	//TEXT N.270
    TEXT271 : BOOL ;	//TEXT N.271
    TEXT272 : BOOL ;	//TEXT N.272
    TEXT257 : BOOL ;	//TEXT N.257
    TEXT258 : BOOL ;	//TEXT N.258
    TEXT259 : BOOL ;	//TEXT N.259
    TEXT260 : BOOL ;	//TEXT N.260
    TEXT261 : BOOL ;	//TEXT N.261
    TEXT262 : BOOL ;	//TEXT N.262
    TEXT263 : BOOL ;	//TEXT N.263
    TEXT264 : BOOL ;	//TEXT N.264
    TEXT281 : BOOL ;	//TEXT N.281
    TEXT282 : BOOL ;	//TEXT N.282
    TEXT283 : BOOL ;	//TEXT N.283
    TEXT284 : BOOL ;	//TEXT N.284
    TEXT285 : BOOL ;	//TEXT N.285
    TEXT286 : BOOL ;	//TEXT N.286
    TEXT287 : BOOL ;	//TEXT N.287
    TEXT288 : BOOL ;	//TEXT N.288
    TEXT273 : BOOL ;	//TEXT N.273
    TEXT274 : BOOL ;	//TEXT N.274
    TEXT275 : BOOL ;	//TEXT N.275
    TEXT276 : BOOL ;	//TEXT N.276
    TEXT277 : BOOL ;	//TEXT N.277
    TEXT278 : BOOL ;	//TEXT N.278
    TEXT279 : BOOL ;	//TEXT N.279
    TEXT280 : BOOL ;	//TEXT N.280
    TEXT297 : BOOL ;	//TEXT N.297
    TEXT298 : BOOL ;	//TEXT N.298
    TEXT299 : BOOL ;	//TEXT N.299
    TEXT300 : BOOL ;	//TEXT N.300
    TEXT301 : BOOL ;	//TEXT N.301
    TEXT302 : BOOL ;	//TEXT N.302
    TEXT303 : BOOL ;	//TEXT N.303
    TEXT304 : BOOL ;	//TEXT N.304
    TEXT289 : BOOL ;	//TEXT N.289
    TEXT290 : BOOL ;	//TEXT N.290
    TEXT291 : BOOL ;	//TEXT N.291
    TEXT292 : BOOL ;	//TEXT N.292
    TEXT293 : BOOL ;	//TEXT N.293
    TEXT294 : BOOL ;	//TEXT N.294
    TEXT295 : BOOL ;	//TEXT N.295
    TEXT296 : BOOL ;	//TEXT N.296
    TEXT313 : BOOL ;	//TEXT N.313
    TEXT314 : BOOL ;	//TEXT N.314
    TEXT315 : BOOL ;	//TEXT N.315
    TEXT316 : BOOL ;	//TEXT N.316
    TEXT317 : BOOL ;	//TEXT N.317
    TEXT318 : BOOL ;	//TEXT N.318
    TEXT319 : BOOL ;	//TEXT N.319
    TEXT320 : BOOL ;	//TEXT N.320
    TEXT305 : BOOL ;	//TEXT N.305
    TEXT306 : BOOL ;	//TEXT N.306
    TEXT307 : BOOL ;	//TEXT N.307
    TEXT308 : BOOL ;	//TEXT N.308
    TEXT309 : BOOL ;	//TEXT N.309
    TEXT310 : BOOL ;	//TEXT N.310
    TEXT311 : BOOL ;	//TEXT N.311
    TEXT312 : BOOL ;	//TEXT N.312
    TEXT329 : BOOL ;
    TEXT330 : BOOL ;
    TEXT331 : BOOL ;
    TEXT332 : BOOL ;
    TEXT333 : BOOL ;
    TEXT334 : BOOL ;
    TEXT335 : BOOL ;
    TEXT336 : BOOL ;
    TEXT321 : BOOL ;
    TEXT322 : BOOL ;
    TEXT323 : BOOL ;
    TEXT324 : BOOL ;
    TEXT325 : BOOL ;
    TEXT326 : BOOL ;
    TEXT327 : BOOL ;
    TEXT328 : BOOL ;
    TEXT345 : BOOL ;
    TEXT346 : BOOL ;
    TEXT347 : BOOL ;
    TEXT348 : BOOL ;
    TEXT349 : BOOL ;
    TEXT350 : BOOL ;
    TEXT351 : BOOL ;
    TEXT352 : BOOL ;
    TEXT337 : BOOL ;
    TEXT338 : BOOL ;
    TEXT339 : BOOL ;
    TEXT340 : BOOL ;
    TEXT341 : BOOL ;
    TEXT342 : BOOL ;
    TEXT343 : BOOL ;
    TEXT344 : BOOL ;
    TEXT361 : BOOL ;	//TEXT N.361
    TEXT362 : BOOL ;	//TEXT N.362
    TEXT363 : BOOL ;	//TEXT N.363
    TEXT364 : BOOL ;	//TEXT N.364
    TEXT365 : BOOL ;	//TEXT N.365
    TEXT366 : BOOL ;	//TEXT N.366
    TEXT367 : BOOL ;	//TEXT N.367
    TEXT368 : BOOL ;	//TEXT N.368
    TEXT353 : BOOL ;	//TEXT N.353
    TEXT354 : BOOL ;	//TEXT N.354
    TEXT355 : BOOL ;	//TEXT N.355
    TEXT356 : BOOL ;	//TEXT N.356
    TEXT357 : BOOL ;	//TEXT N.357
    TEXT358 : BOOL ;	//TEXT N.358
    TEXT359 : BOOL ;	//TEXT N.359
    TEXT360 : BOOL ;	//TEXT N.360
    TEXT377 : BOOL ;	//TEXT N.377
    TEXT378 : BOOL ;	//TEXT N.378
    TEXT379 : BOOL ;	//TEXT N.379
    TEXT380 : BOOL ;	//TEXT N.380
    TEXT381 : BOOL ;	//TEXT N.381
    TEXT382 : BOOL ;	//TEXT N.382
    TEXT383 : BOOL ;	//TEXT N.383
    TEXT384 : BOOL ;	//TEXT N.384
    TEXT369 : BOOL ;	//TEXT N.369
    TEXT370 : BOOL ;	//TEXT N.370
    TEXT371 : BOOL ;	//TEXT N.371
    TEXT372 : BOOL ;	//TEXT N.372
    TEXT373 : BOOL ;	//TEXT N.373
    TEXT374 : BOOL ;	//TEXT N.374
    TEXT375 : BOOL ;	//TEXT N.375
    TEXT376 : BOOL ;	//TEXT N.376
    TEXT393 : BOOL ;	//TEXT N.393
    TEXT394 : BOOL ;	//TEXT N.394
    TEXT395 : BOOL ;	//TEXT N.395
    TEXT396 : BOOL ;	//TEXT N.396
    TEXT397 : BOOL ;	//TEXT N.397
    TEXT398 : BOOL ;	//TEXT N.398
    TEXT399 : BOOL ;	//TEXT N.399
    TEXT400 : BOOL ;	//TEXT N.400
    TEXT385 : BOOL ;	//TEXT N.385
    TEXT386 : BOOL ;	//TEXT N.386
    TEXT387 : BOOL ;	//TEXT N.387
    TEXT388 : BOOL ;	//TEXT N.388
    TEXT389 : BOOL ;	//TEXT N.389
    TEXT390 : BOOL ;	//TEXT N.390
    TEXT391 : BOOL ;	//TEXT N.391
    TEXT392 : BOOL ;	//TEXT N.392
    TEXT409 : BOOL ;	//TEXT N.409
    TEXT410 : BOOL ;	//TEXT N.410
    TEXT411 : BOOL ;	//TEXT N.411
    TEXT412 : BOOL ;	//TEXT N.412
    TEXT413 : BOOL ;	//TEXT N.413
    TEXT414 : BOOL ;	//TEXT N.414
    TEXT415 : BOOL ;	//TEXT N.415
    TEXT416 : BOOL ;	//TEXT N.416
    TEXT401 : BOOL ;	//TEXT N.401
    TEXT402 : BOOL ;	//TEXT N.402
    TEXT403 : BOOL ;	//TEXT N.403
    TEXT404 : BOOL ;	//TEXT N.404
    TEXT405 : BOOL ;	//TEXT N.405
    TEXT406 : BOOL ;	//TEXT N.406
    TEXT407 : BOOL ;	//TEXT N.407
    TEXT408 : BOOL ;	//TEXT N.408
    TEXT425 : BOOL ;	//TEXT N.425
    TEXT426 : BOOL ;	//TEXT N.426
    TEXT427 : BOOL ;	//TEXT N.427
    TEXT428 : BOOL ;	//TEXT N.428
    TEXT429 : BOOL ;	//TEXT N.429
    TEXT430 : BOOL ;	//TEXT N.430
    TEXT431 : BOOL ;	//TEXT N.431
    TEXT432 : BOOL ;	//TEXT N.432
    TEXT417 : BOOL ;	//TEXT N.417
    TEXT418 : BOOL ;	//TEXT N.418
    TEXT419 : BOOL ;	//TEXT N.419
    TEXT420 : BOOL ;	//TEXT N.420
    TEXT421 : BOOL ;	//TEXT N.421
    TEXT422 : BOOL ;	//TEXT N.422
    TEXT423 : BOOL ;	//TEXT N.423
    TEXT424 : BOOL ;	//TEXT N.424
    TEXT441 : BOOL ;	//TEXT N.441
    TEXT442 : BOOL ;	//TEXT N.442
    TEXT443 : BOOL ;	//TEXT N.443
    TEXT444 : BOOL ;	//TEXT N.444
    TEXT445 : BOOL ;	//TEXT N.445
    TEXT446 : BOOL ;	//TEXT N.446
    TEXT447 : BOOL ;	//TEXT N.447
    TEXT448 : BOOL ;	//TEXT N.448
    TEXT433 : BOOL ;	//TEXT N.433
    TEXT434 : BOOL ;	//TEXT N.434
    TEXT435 : BOOL ;	//TEXT N.435
    TEXT436 : BOOL ;	//TEXT N.436
    TEXT437 : BOOL ;	//TEXT N.437
    TEXT438 : BOOL ;	//TEXT N.438
    TEXT439 : BOOL ;	//TEXT N.439
    TEXT440 : BOOL ;	//TEXT N.440
    TEXT457 : BOOL ;	//TEXT N.457
    TEXT458 : BOOL ;	//TEXT N.458
    TEXT459 : BOOL ;	//TEXT N.459
    TEXT460 : BOOL ;	//TEXT N.460
    TEXT461 : BOOL ;	//TEXT N.461
    TEXT462 : BOOL ;	//TEXT N.462
    TEXT463 : BOOL ;	//TEXT N.463
    TEXT464 : BOOL ;	//TEXT N.464
    TEXT449 : BOOL ;	//TEXT N.449
    TEXT450 : BOOL ;	//TEXT N.450
    TEXT451 : BOOL ;	//TEXT N.451
    TEXT452 : BOOL ;	//TEXT N.452
    TEXT453 : BOOL ;	//TEXT N.453
    TEXT454 : BOOL ;	//TEXT N.454
    TEXT455 : BOOL ;	//TEXT N.455
    TEXT456 : BOOL ;	//TEXT N.456
    TEXT473 : BOOL ;	//TEXT N.473
    TEXT474 : BOOL ;	//TEXT N.474
    TEXT475 : BOOL ;	//TEXT N.475
    TEXT476 : BOOL ;	//TEXT N.476
    TEXT477 : BOOL ;	//TEXT N.477
    TEXT478 : BOOL ;	//TEXT N.478
    TEXT479 : BOOL ;	//TEXT N.479
    TEXT480 : BOOL ;	//TEXT N.480
    TEXT465 : BOOL ;	//TEXT N.465
    TEXT466 : BOOL ;	//TEXT N.466
    TEXT467 : BOOL ;	//TEXT N.467
    TEXT468 : BOOL ;	//TEXT N.468
    TEXT469 : BOOL ;	//TEXT N.469
    TEXT470 : BOOL ;	//TEXT N.470
    TEXT471 : BOOL ;	//TEXT N.471
    TEXT472 : BOOL ;	//TEXT N.472
    TEXT489 : BOOL ;	//TEXT N.489
    TEXT490 : BOOL ;	//TEXT N.490
    TEXT491 : BOOL ;	//TEXT N.491
    TEXT492 : BOOL ;	//TEXT N.492
    TEXT493 : BOOL ;	//TEXT N.493
    TEXT494 : BOOL ;	//TEXT N.494
    TEXT495 : BOOL ;	//TEXT N.495
    TEXT496 : BOOL ;	//TEXT N.496
    TEXT481 : BOOL ;	//TEXT N.481
    TEXT482 : BOOL ;	//TEXT N.482
    TEXT483 : BOOL ;	//TEXT N.483
    TEXT484 : BOOL ;	//TEXT N.484
    TEXT485 : BOOL ;	//TEXT N.485
    TEXT486 : BOOL ;	//TEXT N.486
    TEXT487 : BOOL ;	//TEXT N.487
    TEXT488 : BOOL ;	//TEXT N.488
    TEXT505 : BOOL ;	//TEXT N.505
    TEXT506 : BOOL ;	//TEXT N.506
    TEXT507 : BOOL ;	//TEXT N.507
    TEXT508 : BOOL ;	//TEXT N.508
    TEXT509 : BOOL ;	//TEXT N.509
    TEXT510 : BOOL ;	//TEXT N.510
    TEXT511 : BOOL ;	//TEXT N.511
    TEXT512 : BOOL ;	//TEXT N.512
    TEXT497 : BOOL ;	//TEXT N.497
    TEXT498 : BOOL ;	//TEXT N.498
    TEXT499 : BOOL ;	//TEXT N.499
    TEXT500 : BOOL ;	//TEXT N.500
    TEXT501 : BOOL ;	//TEXT N.501
    TEXT502 : BOOL ;	//TEXT N.502
    TEXT503 : BOOL ;	//TEXT N.503
    TEXT504 : BOOL ;	//TEXT N.504
    TEXT521 : BOOL ;	//TEXT N.521
    TEXT522 : BOOL ;	//TEXT N.522
    TEXT523 : BOOL ;	//TEXT N.523
    TEXT524 : BOOL ;	//TEXT N.524
    TEXT525 : BOOL ;	//TEXT N.525
    TEXT526 : BOOL ;	//TEXT N.526
    TEXT527 : BOOL ;	//TEXT N.527
    TEXT528 : BOOL ;	//TEXT N.528
    TEXT513 : BOOL ;	//TEXT N.513
    TEXT514 : BOOL ;	//TEXT N.514
    TEXT515 : BOOL ;	//TEXT N.515
    TEXT516 : BOOL ;	//TEXT N.516
    TEXT517 : BOOL ;	//TEXT N.517
    TEXT518 : BOOL ;	//TEXT N.518
    TEXT519 : BOOL ;	//TEXT N.519
    TEXT520 : BOOL ;	//TEXT N.520
    TEXT537 : BOOL ;	//TEXT N.537
    TEXT538 : BOOL ;	//TEXT N.538
    TEXT539 : BOOL ;	//TEXT N.539
    TEXT540 : BOOL ;	//TEXT N.540
    TEXT541 : BOOL ;	//TEXT N.541
    TEXT542 : BOOL ;	//TEXT N.542
    TEXT543 : BOOL ;	//TEXT N.543
    TEXT544 : BOOL ;	//TEXT N.544
    TEXT529 : BOOL ;	//TEXT N.529
    TEXT530 : BOOL ;	//TEXT N.530
    TEXT531 : BOOL ;	//TEXT N.531
    TEXT532 : BOOL ;	//TEXT N.532
    TEXT533 : BOOL ;	//TEXT N.533
    TEXT534 : BOOL ;	//TEXT N.534
    TEXT535 : BOOL ;	//TEXT N.535
    TEXT536 : BOOL ;	//TEXT N.536
    TEXT553 : BOOL ;	//TEXT N.553
    TEXT554 : BOOL ;	//TEXT N.554
    TEXT555 : BOOL ;	//TEXT N.555
    TEXT556 : BOOL ;	//TEXT N.556
    TEXT557 : BOOL ;	//TEXT N.557
    TEXT558 : BOOL ;	//TEXT N.558
    TEXT559 : BOOL ;	//TEXT N.559
    TEXT560 : BOOL ;	//TEXT N.560
    TEXT545 : BOOL ;	//TEXT N.545
    TEXT546 : BOOL ;	//TEXT N.546
    TEXT547 : BOOL ;	//TEXT N.547
    TEXT548 : BOOL ;	//TEXT N.548
    TEXT549 : BOOL ;	//TEXT N.549
    TEXT550 : BOOL ;	//TEXT N.550
    TEXT551 : BOOL ;	//TEXT N.551
    TEXT552 : BOOL ;	//TEXT N.552
    TEXT569 : BOOL ;	//TEXT N.569
    TEXT570 : BOOL ;	//TEXT N.570
    TEXT571 : BOOL ;	//TEXT N.571
    TEXT572 : BOOL ;	//TEXT N.572
    TEXT573 : BOOL ;	//TEXT N.573
    TEXT574 : BOOL ;	//TEXT N.574
    TEXT575 : BOOL ;	//TEXT N.575
    TEXT576 : BOOL ;	//TEXT N.576
    TEXT561 : BOOL ;	//TEXT N.561
    TEXT562 : BOOL ;	//TEXT N.562
    TEXT563 : BOOL ;	//TEXT N.563
    TEXT564 : BOOL ;	//TEXT N.564
    TEXT565 : BOOL ;	//TEXT N.565
    TEXT566 : BOOL ;	//TEXT N.566
    TEXT567 : BOOL ;	//TEXT N.567
    TEXT568 : BOOL ;	//TEXT N.568
    TEXT585 : BOOL ;	//TEXT N.585
    TEXT586 : BOOL ;	//TEXT N.586
    TEXT587 : BOOL ;	//TEXT N.587
    TEXT588 : BOOL ;	//TEXT N.588
    TEXT589 : BOOL ;	//TEXT N.589
    TEXT590 : BOOL ;	//TEXT N.590
    TEXT591 : BOOL ;	//TEXT N.591
    TEXT592 : BOOL ;	//TEXT N.592
    TEXT577 : BOOL ;	//TEXT N.577
    TEXT578 : BOOL ;	//TEXT N.578
    TEXT579 : BOOL ;	//TEXT N.579
    TEXT580 : BOOL ;	//TEXT N.580
    TEXT581 : BOOL ;	//TEXT N.581
    TEXT582 : BOOL ;	//TEXT N.582
    TEXT583 : BOOL ;	//TEXT N.583
    TEXT584 : BOOL ;	//TEXT N.584
    TEXT601 : BOOL ;	//TEXT N.601
    TEXT602 : BOOL ;	//TEXT N.602
    TEXT603 : BOOL ;	//TEXT N.603
    TEXT604 : BOOL ;	//TEXT N.604
    TEXT605 : BOOL ;	//TEXT N.605
    TEXT606 : BOOL ;	//TEXT N.606
    TEXT607 : BOOL ;	//TEXT N.607
    TEXT608 : BOOL ;	//TEXT N.608
    TEXT593 : BOOL ;	//TEXT N.593
    TEXT594 : BOOL ;	//TEXT N.594
    TEXT595 : BOOL ;	//TEXT N.595
    TEXT596 : BOOL ;	//TEXT N.596
    TEXT597 : BOOL ;	//TEXT N.597
    TEXT598 : BOOL ;	//TEXT N.598
    TEXT599 : BOOL ;	//TEXT N.599
    TEXT600 : BOOL ;	//TEXT N.600
    TEXT617 : BOOL ;	//TEXT N.617
    TEXT618 : BOOL ;	//TEXT N.618
    TEXT619 : BOOL ;	//TEXT N.619
    TEXT620 : BOOL ;	//TEXT N.620
    TEXT621 : BOOL ;	//TEXT N.621
    TEXT622 : BOOL ;	//TEXT N.622
    TEXT623 : BOOL ;	//TEXT N.623
    TEXT624 : BOOL ;	//TEXT N.624
    TEXT609 : BOOL ;	//TEXT N.609
    TEXT610 : BOOL ;	//TEXT N.610
    TEXT611 : BOOL ;	//TEXT N.611
    TEXT612 : BOOL ;	//TEXT N.612
    TEXT613 : BOOL ;	//TEXT N.613
    TEXT614 : BOOL ;	//TEXT N.614
    TEXT615 : BOOL ;	//TEXT N.615
    TEXT616 : BOOL ;	//TEXT N.616
    TEXT633 : BOOL ;	//TEXT N.633
    TEXT634 : BOOL ;	//TEXT N.634
    TEXT635 : BOOL ;	//TEXT N.635
    TEXT636 : BOOL ;	//TEXT N.636
    TEXT637 : BOOL ;	//TEXT N.637
    TEXT638 : BOOL ;	//TEXT N.638
    TEXT639 : BOOL ;	//TEXT N.639
    TEXT640 : BOOL ;	//TEXT N.640
    TEXT625 : BOOL ;	//TEXT N.625
    TEXT626 : BOOL ;	//TEXT N.626
    TEXT627 : BOOL ;	//TEXT N.627
    TEXT628 : BOOL ;	//TEXT N.628
    TEXT629 : BOOL ;	//TEXT N.629
    TEXT630 : BOOL ;	//TEXT N.630
    TEXT631 : BOOL ;	//TEXT N.631
    TEXT632 : BOOL ;	//TEXT N.632
   END_STRUCT ;
   SegnalazioniAllarme : STRUCT
    TEXT9 : BOOL ;
    TEXT10 : BOOL ;
    TEXT11 : BOOL ;
    TEXT12 : BOOL ;
    TEXT13 : BOOL ;
    TEXT14 : BOOL ;
    TEXT15 : BOOL ;
    TEXT16 : BOOL ;
    TEXT1 : BOOL ;
    TEXT2 : BOOL ;
    TEXT3 : BOOL ;
    TEXT4 : BOOL ;
    TEXT5 : BOOL ;
    TEXT6 : BOOL ;
    TEXT7 : BOOL ;
    TEXT8 : BOOL ;
    TEXT25 : BOOL ;
    TEXT26 : BOOL ;
    TEXT27 : BOOL ;
    TEXT28 : BOOL ;
    TEXT29 : BOOL ;
    TEXT30 : BOOL ;
    TEXT31 : BOOL ;
    TEXT32 : BOOL ;
    TEXT17 : BOOL ;
    TEXT18 : BOOL ;
    TEXT19 : BOOL ;
    TEXT20 : BOOL ;
    TEXT21 : BOOL ;
    TEXT22 : BOOL ;
    TEXT23 : BOOL ;
    TEXT24 : BOOL ;
    TEXT41 : BOOL ;
    TEXT42 : BOOL ;
    TEXT43 : BOOL ;
    TEXT44 : BOOL ;
    TEXT45 : BOOL ;
    TEXT46 : BOOL ;
    TEXT47 : BOOL ;
    TEXT48 : BOOL ;
    TEXT33 : BOOL ;
    TEXT34 : BOOL ;
    TEXT35 : BOOL ;
    TEXT36 : BOOL ;
    TEXT37 : BOOL ;
    TEXT38 : BOOL ;
    TEXT39 : BOOL ;
    TEXT40 : BOOL ;
    TEXT57 : BOOL ;	//TEXT N.57
    TEXT58 : BOOL ;	//TEXT N.58
    TEXT59 : BOOL ;	//TEXT N.59
    TEXT60 : BOOL ;	//TEXT N.60
    TEXT61 : BOOL ;	//TEXT N.61
    TEXT62 : BOOL ;	//TEXT N.62
    TEXT63 : BOOL ;	//TEXT N.63
    TEXT64 : BOOL ;	//TEXT N.64
    TEXT49 : BOOL ;	//TEXT N.49
    TEXT50 : BOOL ;	//TEXT N.50
    TEXT51 : BOOL ;	//TEXT N.51
    TEXT52 : BOOL ;	//TEXT N.52
    TEXT53 : BOOL ;	//TEXT N.53
    TEXT54 : BOOL ;	//TEXT N.54
    TEXT55 : BOOL ;	//TEXT N.55
    TEXT56 : BOOL ;	//TEXT N.56
    TEXT73 : BOOL ;
    TEXT74 : BOOL ;
    TEXT75 : BOOL ;
    TEXT76 : BOOL ;
    TEXT77 : BOOL ;	//TEXT N.77
    TEXT78 : BOOL ;	//TEXT N.78
    TEXT79 : BOOL ;	//TEXT N.79
    TEXT80 : BOOL ;	//TEXT N.80
    TEXT65 : BOOL ;	//TEXT N.65
    TEXT66 : BOOL ;	//TEXT N.66
    TEXT67 : BOOL ;	//TEXT N.67
    TEXT68 : BOOL ;	//TEXT N.68
    TEXT69 : BOOL ;	//TEXT N.69
    TEXT70 : BOOL ;	//TEXT N.70
    TEXT71 : BOOL ;	//TEXT N.71
    TEXT72 : BOOL ;	//TEXT N.72
    TEXT89 : BOOL ;
    TEXT90 : BOOL ;
    TEXT91 : BOOL ;
    TEXT92 : BOOL ;
    TEXT93 : BOOL ;	//TEXT N.93
    TEXT94 : BOOL ;	//TEXT N.94
    TEXT95 : BOOL ;	//TEXT N.95
    TEXT96 : BOOL ;	//TEXT N.96
    TEXT81 : BOOL ;	//TEXT N.81
    TEXT82 : BOOL ;	//TEXT N.82
    TEXT83 : BOOL ;	//TEXT N.83
    TEXT84 : BOOL ;	//TEXT N.84
    TEXT85 : BOOL ;	//TEXT N.85
    TEXT86 : BOOL ;	//TEXT N.86
    TEXT87 : BOOL ;	//TEXT N.87
    TEXT88 : BOOL ;	//TEXT N.88
    TEXT105 : BOOL ;	//TEXT N.105
    TEXT106 : BOOL ;	//TEXT N.106
    TEXT107 : BOOL ;	//TEXT N.107
    TEXT108 : BOOL ;	//TEXT N.108
    TEXT109 : BOOL ;	//TEXT N.109
    TEXT110 : BOOL ;	//TEXT N.110
    TEXT111 : BOOL ;	//TEXT N.111
    TEXT112 : BOOL ;	//TEXT N.112
    TEXT97 : BOOL ;	//TEXT N.17
    TEXT98 : BOOL ;	//TEXT N.18
    TEXT99 : BOOL ;	//TEXT N.19
    TEXT100 : BOOL ;	//TEXT N.100
    TEXT101 : BOOL ;	//TEXT N.101
    TEXT102 : BOOL ;	//TEXT N.102
    TEXT103 : BOOL ;	//TEXT N.103
    TEXT104 : BOOL ;	//TEXT N.104
    TEXT121 : BOOL ;	//TEXT N.121
    TEXT122 : BOOL ;	//TEXT N.122
    TEXT123 : BOOL ;	//TEXT N.123
    TEXT124 : BOOL ;	//TEXT N.124
    TEXT125 : BOOL ;	//TEXT N.125
    TEXT126 : BOOL ;	//TEXT N.126
    TEXT127 : BOOL ;	//TEXT N.127
    TEXT128 : BOOL ;	//TEXT N.128
    TEXT113 : BOOL ;	//TEXT N.113
    TEXT114 : BOOL ;	//TEXT N.114
    TEXT115 : BOOL ;	//TEXT N.115
    TEXT116 : BOOL ;	//TEXT N.116
    TEXT117 : BOOL ;	//TEXT N.117
    TEXT118 : BOOL ;	//TEXT N.118
    TEXT119 : BOOL ;	//TEXT N.119
    TEXT120 : BOOL ;	//TEXT N.120
    TEXT137 : BOOL ;	//TEXT N.137
    TEXT138 : BOOL ;	//TEXT N.138
    TEXT139 : BOOL ;	//TEXT N.139
    TEXT140 : BOOL ;	//TEXT N.140
    TEXT141 : BOOL ;	//TEXT N.141
    TEXT142 : BOOL ;	//TEXT N.142
    TEXT143 : BOOL ;	//TEXT N.143
    TEXT144 : BOOL ;	//TEXT N.144
    TEXT129 : BOOL ;	//TEXT N.129
    TEXT130 : BOOL ;	//TEXT N.130
    TEXT131 : BOOL ;	//TEXT N.131
    TEXT132 : BOOL ;	//TEXT N.132
    TEXT133 : BOOL ;	//TEXT N.133
    TEXT134 : BOOL ;	//TEXT N.134
    TEXT135 : BOOL ;	//TEXT N.135
    TEXT136 : BOOL ;	//TEXT N.136
    TEXT153 : BOOL ;	//TEXT N.153
    TEXT154 : BOOL ;	//TEXT N.154
    TEXT155 : BOOL ;	//TEXT N.155
    TEXT156 : BOOL ;	//TEXT N.156
    TEXT157 : BOOL ;	//TEXT N.157
    TEXT158 : BOOL ;	//TEXT N.158
    TEXT159 : BOOL ;	//TEXT N.159
    TEXT160 : BOOL ;	//TEXT N.160
    TEXT145 : BOOL ;	//TEXT N.145
    TEXT146 : BOOL ;	//TEXT N.146
    TEXT147 : BOOL ;	//TEXT N.147
    TEXT148 : BOOL ;	//TEXT N.148
    TEXT149 : BOOL ;	//TEXT N.149
    TEXT150 : BOOL ;	//TEXT N.150
    TEXT151 : BOOL ;	//TEXT N.151
    TEXT152 : BOOL ;	//TEXT N.152
    TEXT169 : BOOL ;	//TEXT N.169
    TEXT170 : BOOL ;	//TEXT N.170
    TEXT171 : BOOL ;	//TEXT N.171
    TEXT172 : BOOL ;	//TEXT N.172
    TEXT173 : BOOL ;	//TEXT N.173
    TEXT174 : BOOL ;	//TEXT N.174
    TEXT175 : BOOL ;	//TEXT N.175
    TEXT176 : BOOL ;	//TEXT N.176
    TEXT161 : BOOL ;	//TEXT N.161
    TEXT162 : BOOL ;	//TEXT N.162
    TEXT163 : BOOL ;	//TEXT N.163
    TEXT164 : BOOL ;	//TEXT N.164
    TEXT165 : BOOL ;	//TEXT N.165
    TEXT166 : BOOL ;	//TEXT N.166
    TEXT167 : BOOL ;	//TEXT N.167
    TEXT168 : BOOL ;	//TEXT N.168
    TEXT185 : BOOL ;	//TEXT N.185
    TEXT186 : BOOL ;	//TEXT N.186
    TEXT187 : BOOL ;	//TEXT N.187
    TEXT188 : BOOL ;	//TEXT N.188
    TEXT189 : BOOL ;	//TEXT N.189
    TEXT190 : BOOL ;	//TEXT N.190
    TEXT191 : BOOL ;	//TEXT N.191
    TEXT192 : BOOL ;	//TEXT N.192
    TEXT177 : BOOL ;	//TEXT N.177
    TEXT178 : BOOL ;	//TEXT N.178
    TEXT179 : BOOL ;	//TEXT N.179
    TEXT180 : BOOL ;	//TEXT N.180
    TEXT181 : BOOL ;	//TEXT N.181
    TEXT182 : BOOL ;	//TEXT N.182
    TEXT183 : BOOL ;	//TEXT N.183
    TEXT184 : BOOL ;	//TEXT N.184
    TEXT201 : BOOL ;	//TEXT N.201
    TEXT202 : BOOL ;	//TEXT N.202
    TEXT203 : BOOL ;	//TEXT N.203
    TEXT204 : BOOL ;	//TEXT N.204
    TEXT205 : BOOL ;	//TEXT N.205
    TEXT206 : BOOL ;	//TEXT N.206
    TEXT207 : BOOL ;	//TEXT N.207
    TEXT208 : BOOL ;	//TEXT N.208
    TEXT193 : BOOL ;	//TEXT N.193
    TEXT194 : BOOL ;	//TEXT N.194
    TEXT195 : BOOL ;	//TEXT N.195
    TEXT196 : BOOL ;	//TEXT N.196
    TEXT197 : BOOL ;	//TEXT N.197
    TEXT198 : BOOL ;	//TEXT N.198
    TEXT199 : BOOL ;	//TEXT N.199
    TEXT200 : BOOL ;	//TEXT N.200
    TEXT217 : BOOL ;	//TEXT N.217
    TEXT218 : BOOL ;	//TEXT N.218
    TEXT219 : BOOL ;	//TEXT N.219
    TEXT220 : BOOL ;	//TEXT N.220
    TEXT221 : BOOL ;	//TEXT N.221
    TEXT222 : BOOL ;	//TEXT N.222
    TEXT223 : BOOL ;	//TEXT N.223
    TEXT224 : BOOL ;	//TEXT N.224
    TEXT209 : BOOL ;	//TEXT N.209
    TEXT210 : BOOL ;	//TEXT N.210
    TEXT211 : BOOL ;	//TEXT N.211
    TEXT212 : BOOL ;	//TEXT N.212
    TEXT213 : BOOL ;	//TEXT N.213
    TEXT214 : BOOL ;	//TEXT N.214
    TEXT215 : BOOL ;	//TEXT N.215
    TEXT216 : BOOL ;	//TEXT N.216
    TEXT233 : BOOL ;	//TEXT N.233
    TEXT234 : BOOL ;	//TEXT N.234
    TEXT235 : BOOL ;	//TEXT N.235
    TEXT236 : BOOL ;	//TEXT N.236
    TEXT237 : BOOL ;	//TEXT N.237
    TEXT238 : BOOL ;	//TEXT N.238
    TEXT239 : BOOL ;	//TEXT N.239
    TEXT240 : BOOL ;	//TEXT N.240
    TEXT225 : BOOL ;	//TEXT N.225
    TEXT226 : BOOL ;	//TEXT N.226
    TEXT227 : BOOL ;	//TEXT N.227
    TEXT228 : BOOL ;	//TEXT N.228
    TEXT229 : BOOL ;	//TEXT N.229
    TEXT230 : BOOL ;	//TEXT N.230
    TEXT231 : BOOL ;	//TEXT N.231
    TEXT232 : BOOL ;	//TEXT N.232
    TEXT249 : BOOL ;	//TEXT N.249
    TEXT250 : BOOL ;	//TEXT N.250
    TEXT251 : BOOL ;	//TEXT N.251
    TEXT252 : BOOL ;	//TEXT N.252
    TEXT253 : BOOL ;	//TEXT N.253
    TEXT254 : BOOL ;	//TEXT N.254
    TEXT255 : BOOL ;	//TEXT N.255
    TEXT256 : BOOL ;	//TEXT N.256
    TEXT241 : BOOL ;	//TEXT N.241
    TEXT242 : BOOL ;	//TEXT N.242
    TEXT243 : BOOL ;	//TEXT N.243
    TEXT244 : BOOL ;	//TEXT N.244
    TEXT245 : BOOL ;	//TEXT N.245
    TEXT246 : BOOL ;	//TEXT N.246
    TEXT247 : BOOL ;	//TEXT N.247
    TEXT248 : BOOL ;	//TEXT N.248
    TEXT265 : BOOL ;	//TEXT N.265
    TEXT266 : BOOL ;	//TEXT N.266
    TEXT267 : BOOL ;	//TEXT N.267
    TEXT268 : BOOL ;	//TEXT N.268
    TEXT269 : BOOL ;	//TEXT N.269
    TEXT270 : BOOL ;	//TEXT N.270
    TEXT271 : BOOL ;	//TEXT N.271
    TEXT272 : BOOL ;	//TEXT N.272
    TEXT257 : BOOL ;	//TEXT N.257
    TEXT258 : BOOL ;	//TEXT N.258
    TEXT259 : BOOL ;	//TEXT N.259
    TEXT260 : BOOL ;	//TEXT N.260
    TEXT261 : BOOL ;	//TEXT N.261
    TEXT262 : BOOL ;	//TEXT N.262
    TEXT263 : BOOL ;	//TEXT N.263
    TEXT264 : BOOL ;	//TEXT N.264
    TEXT281 : BOOL ;	//TEXT N.281
    TEXT282 : BOOL ;	//TEXT N.282
    TEXT283 : BOOL ;	//TEXT N.283
    TEXT284 : BOOL ;	//TEXT N.284
    TEXT285 : BOOL ;	//TEXT N.285
    TEXT286 : BOOL ;	//TEXT N.286
    TEXT287 : BOOL ;	//TEXT N.287
    TEXT288 : BOOL ;	//TEXT N.288
    TEXT273 : BOOL ;	//TEXT N.273
    TEXT274 : BOOL ;	//TEXT N.274
    TEXT275 : BOOL ;	//TEXT N.275
    TEXT276 : BOOL ;	//TEXT N.276
    TEXT277 : BOOL ;	//TEXT N.277
    TEXT278 : BOOL ;	//TEXT N.278
    TEXT279 : BOOL ;	//TEXT N.279
    TEXT280 : BOOL ;	//TEXT N.280
    TEXT297 : BOOL ;	//TEXT N.297
    TEXT298 : BOOL ;	//TEXT N.298
    TEXT299 : BOOL ;	//TEXT N.299
    TEXT300 : BOOL ;	//TEXT N.300
    TEXT301 : BOOL ;	//TEXT N.301
    TEXT302 : BOOL ;	//TEXT N.302
    TEXT303 : BOOL ;	//TEXT N.303
    TEXT304 : BOOL ;	//TEXT N.304
    TEXT289 : BOOL ;	//TEXT N.289
    TEXT290 : BOOL ;	//TEXT N.290
    TEXT291 : BOOL ;	//TEXT N.291
    TEXT292 : BOOL ;	//TEXT N.292
    TEXT293 : BOOL ;	//TEXT N.293
    TEXT294 : BOOL ;	//TEXT N.294
    TEXT295 : BOOL ;	//TEXT N.295
    TEXT296 : BOOL ;	//TEXT N.296
    TEXT313 : BOOL ;	//TEXT N.313
    TEXT314 : BOOL ;	//TEXT N.314
    TEXT315 : BOOL ;	//TEXT N.315
    TEXT316 : BOOL ;	//TEXT N.316
    TEXT317 : BOOL ;	//TEXT N.317
    TEXT318 : BOOL ;	//TEXT N.318
    TEXT319 : BOOL ;	//TEXT N.319
    TEXT320 : BOOL ;	//TEXT N.320
    TEXT305 : BOOL ;	//TEXT N.305
    TEXT306 : BOOL ;	//TEXT N.306
    TEXT307 : BOOL ;	//TEXT N.307
    TEXT308 : BOOL ;	//TEXT N.308
    TEXT309 : BOOL ;	//TEXT N.309
    TEXT310 : BOOL ;	//TEXT N.310
    TEXT311 : BOOL ;	//TEXT N.311
    TEXT312 : BOOL ;	//TEXT N.312
    TEXT329 : BOOL ;	//TEXT N.329
    TEXT330 : BOOL ;	//TEXT N.330
    TEXT331 : BOOL ;	//TEXT N.331
    TEXT332 : BOOL ;	//TEXT N.332
    TEXT333 : BOOL ;	//TEXT N.333
    TEXT334 : BOOL ;	//TEXT N.334
    TEXT335 : BOOL ;	//TEXT N.335
    TEXT336 : BOOL ;	//TEXT N.336
    TEXT321 : BOOL ;	//TEXT N.321
    TEXT322 : BOOL ;	//TEXT N.322
    TEXT323 : BOOL ;	//TEXT N.323
    TEXT324 : BOOL ;	//TEXT N.324
    TEXT325 : BOOL ;	//TEXT N.325
    TEXT326 : BOOL ;	//TEXT N.326
    TEXT327 : BOOL ;	//TEXT N.327
    TEXT328 : BOOL ;	//TEXT N.328
    TEXT345 : BOOL ;	//TEXT N.345
    TEXT346 : BOOL ;	//TEXT N.346
    TEXT347 : BOOL ;	//TEXT N.347
    TEXT348 : BOOL ;	//TEXT N.348
    TEXT349 : BOOL ;	//TEXT N.349
    TEXT350 : BOOL ;	//TEXT N.350
    TEXT351 : BOOL ;	//TEXT N.351
    TEXT352 : BOOL ;	//TEXT N.352
    TEXT337 : BOOL ;	//TEXT N.337
    TEXT338 : BOOL ;	//TEXT N.338
    TEXT339 : BOOL ;	//TEXT N.339
    TEXT340 : BOOL ;	//TEXT N.340
    TEXT341 : BOOL ;	//TEXT N.341
    TEXT342 : BOOL ;	//TEXT N.342
    TEXT343 : BOOL ;	//TEXT N.343
    TEXT344 : BOOL ;	//TEXT N.344
    TEXT361 : BOOL ;	//TEXT N.361
    TEXT362 : BOOL ;	//TEXT N.362
    TEXT363 : BOOL ;	//TEXT N.363
    TEXT364 : BOOL ;	//TEXT N.364
    TEXT365 : BOOL ;	//TEXT N.365
    TEXT366 : BOOL ;	//TEXT N.366
    TEXT367 : BOOL ;	//TEXT N.367
    TEXT368 : BOOL ;	//TEXT N.368
    TEXT353 : BOOL ;	//TEXT N.353
    TEXT354 : BOOL ;	//TEXT N.354
    TEXT355 : BOOL ;	//TEXT N.355
    TEXT356 : BOOL ;	//TEXT N.356
    TEXT357 : BOOL ;	//TEXT N.357
    TEXT358 : BOOL ;	//TEXT N.358
    TEXT359 : BOOL ;	//TEXT N.359
    TEXT360 : BOOL ;	//TEXT N.360
    TEXT377 : BOOL ;	//TEXT N.377
    TEXT378 : BOOL ;	//TEXT N.378
    TEXT379 : BOOL ;	//TEXT N.379
    TEXT380 : BOOL ;	//TEXT N.380
    TEXT381 : BOOL ;	//TEXT N.381
    TEXT382 : BOOL ;	//TEXT N.382
    TEXT383 : BOOL ;	//TEXT N.383
    TEXT384 : BOOL ;	//TEXT N.384
    TEXT369 : BOOL ;	//TEXT N.369
    TEXT370 : BOOL ;	//TEXT N.370
    TEXT371 : BOOL ;	//TEXT N.371
    TEXT372 : BOOL ;	//TEXT N.372
    TEXT373 : BOOL ;	//TEXT N.373
    TEXT374 : BOOL ;	//TEXT N.374
    TEXT375 : BOOL ;	//TEXT N.375
    TEXT376 : BOOL ;	//TEXT N.376
    TEXT393 : BOOL ;	//TEXT N.393
    TEXT394 : BOOL ;	//TEXT N.394
    TEXT395 : BOOL ;	//TEXT N.395
    TEXT396 : BOOL ;	//TEXT N.396
    TEXT397 : BOOL ;	//TEXT N.397
    TEXT398 : BOOL ;	//TEXT N.398
    TEXT399 : BOOL ;	//TEXT N.399
    TEXT400 : BOOL ;	//TEXT N.400
    TEXT385 : BOOL ;	//TEXT N.385
    TEXT386 : BOOL ;	//TEXT N.386
    TEXT387 : BOOL ;	//TEXT N.387
    TEXT388 : BOOL ;	//TEXT N.388
    TEXT389 : BOOL ;	//TEXT N.389
    TEXT390 : BOOL ;	//TEXT N.390
    TEXT391 : BOOL ;	//TEXT N.391
    TEXT392 : BOOL ;	//TEXT N.392
    TEXT409 : BOOL ;	//TEXT N.409
    TEXT410 : BOOL ;	//TEXT N.410
    TEXT411 : BOOL ;	//TEXT N.411
    TEXT412 : BOOL ;	//TEXT N.412
    TEXT413 : BOOL ;	//TEXT N.413
    TEXT414 : BOOL ;	//TEXT N.414
    TEXT415 : BOOL ;	//TEXT N.415
    TEXT416 : BOOL ;	//TEXT N.416
    TEXT401 : BOOL ;	//TEXT N.401
    TEXT402 : BOOL ;	//TEXT N.402
    TEXT403 : BOOL ;	//TEXT N.403
    TEXT404 : BOOL ;	//TEXT N.404
    TEXT405 : BOOL ;	//TEXT N.405
    TEXT406 : BOOL ;	//TEXT N.406
    TEXT407 : BOOL ;	//TEXT N.407
    TEXT408 : BOOL ;	//TEXT N.408
    TEXT425 : BOOL ;	//TEXT N.425
    TEXT426 : BOOL ;	//TEXT N.426
    TEXT427 : BOOL ;	//TEXT N.427
    TEXT428 : BOOL ;	//TEXT N.428
    TEXT429 : BOOL ;	//TEXT N.429
    TEXT430 : BOOL ;	//TEXT N.430
    TEXT431 : BOOL ;	//TEXT N.431
    TEXT432 : BOOL ;	//TEXT N.432
    TEXT417 : BOOL ;	//TEXT N.417
    TEXT418 : BOOL ;	//TEXT N.418
    TEXT419 : BOOL ;	//TEXT N.419
    TEXT420 : BOOL ;	//TEXT N.420
    TEXT421 : BOOL ;	//TEXT N.421
    TEXT422 : BOOL ;	//TEXT N.422
    TEXT423 : BOOL ;	//TEXT N.423
    TEXT424 : BOOL ;	//TEXT N.424
    TEXT441 : BOOL ;	//TEXT N.441
    TEXT442 : BOOL ;	//TEXT N.442
    TEXT443 : BOOL ;	//TEXT N.443
    TEXT444 : BOOL ;	//TEXT N.444
    TEXT445 : BOOL ;	//TEXT N.445
    TEXT446 : BOOL ;	//TEXT N.446
    TEXT447 : BOOL ;	//TEXT N.447
    TEXT448 : BOOL ;	//TEXT N.448
    TEXT433 : BOOL ;	//TEXT N.433
    TEXT434 : BOOL ;	//TEXT N.434
    TEXT435 : BOOL ;	//TEXT N.435
    TEXT436 : BOOL ;	//TEXT N.436
    TEXT437 : BOOL ;	//TEXT N.437
    TEXT438 : BOOL ;	//TEXT N.438
    TEXT439 : BOOL ;	//TEXT N.439
    TEXT440 : BOOL ;	//TEXT N.440
    TEXT457 : BOOL ;	//TEXT N.457
    TEXT458 : BOOL ;	//TEXT N.458
    TEXT459 : BOOL ;	//TEXT N.459
    TEXT460 : BOOL ;	//TEXT N.460
    TEXT461 : BOOL ;	//TEXT N.461
    TEXT462 : BOOL ;	//TEXT N.462
    TEXT463 : BOOL ;	//TEXT N.463
    TEXT464 : BOOL ;	//TEXT N.464
    TEXT449 : BOOL ;	//TEXT N.449
    TEXT450 : BOOL ;	//TEXT N.450
    TEXT451 : BOOL ;	//TEXT N.451
    TEXT452 : BOOL ;	//TEXT N.452
    TEXT453 : BOOL ;	//TEXT N.453
    TEXT454 : BOOL ;	//TEXT N.454
    TEXT455 : BOOL ;	//TEXT N.455
    TEXT456 : BOOL ;	//TEXT N.456
    TEXT473 : BOOL ;	//TEXT N.473
    TEXT474 : BOOL ;	//TEXT N.474
    TEXT475 : BOOL ;	//TEXT N.475
    TEXT476 : BOOL ;	//TEXT N.476
    TEXT477 : BOOL ;	//TEXT N.477
    TEXT478 : BOOL ;	//TEXT N.478
    TEXT479 : BOOL ;	//TEXT N.479
    TEXT480 : BOOL ;	//TEXT N.480
    TEXT465 : BOOL ;	//TEXT N.465
    TEXT466 : BOOL ;	//TEXT N.466
    TEXT467 : BOOL ;	//TEXT N.467
    TEXT468 : BOOL ;	//TEXT N.468
    TEXT469 : BOOL ;	//TEXT N.469
    TEXT470 : BOOL ;	//TEXT N.470
    TEXT471 : BOOL ;	//TEXT N.471
    TEXT472 : BOOL ;	//TEXT N.472
    TEXT489 : BOOL ;	//TEXT N.489
    TEXT490 : BOOL ;	//TEXT N.490
    TEXT491 : BOOL ;	//TEXT N.491
    TEXT492 : BOOL ;	//TEXT N.492
    TEXT493 : BOOL ;	//TEXT N.493
    TEXT494 : BOOL ;	//TEXT N.494
    TEXT495 : BOOL ;	//TEXT N.495
    TEXT496 : BOOL ;	//TEXT N.496
    TEXT481 : BOOL ;	//TEXT N.481
    TEXT482 : BOOL ;	//TEXT N.482
    TEXT483 : BOOL ;	//TEXT N.483
    TEXT484 : BOOL ;	//TEXT N.484
    TEXT485 : BOOL ;	//TEXT N.485
    TEXT486 : BOOL ;	//TEXT N.486
    TEXT487 : BOOL ;	//TEXT N.487
    TEXT488 : BOOL ;	//TEXT N.488
    TEXT505 : BOOL ;	//TEXT N.505
    TEXT506 : BOOL ;	//TEXT N.506
    TEXT507 : BOOL ;	//TEXT N.507
    TEXT508 : BOOL ;	//TEXT N.508
    TEXT509 : BOOL ;	//TEXT N.509
    TEXT510 : BOOL ;	//TEXT N.510
    TEXT511 : BOOL ;	//TEXT N.511
    TEXT512 : BOOL ;	//TEXT N.512
    TEXT497 : BOOL ;	//TEXT N.497
    TEXT498 : BOOL ;	//TEXT N.498
    TEXT499 : BOOL ;	//TEXT N.499
    TEXT500 : BOOL ;	//TEXT N.500
    TEXT501 : BOOL ;	//TEXT N.501
    TEXT502 : BOOL ;	//TEXT N.502
    TEXT503 : BOOL ;	//TEXT N.503
    TEXT504 : BOOL ;	//TEXT N.504
    TEXT521 : BOOL ;	//TEXT N.521
    TEXT522 : BOOL ;	//TEXT N.522
    TEXT523 : BOOL ;	//TEXT N.523
    TEXT524 : BOOL ;	//TEXT N.524
    TEXT525 : BOOL ;	//TEXT N.525
    TEXT526 : BOOL ;	//TEXT N.526
    TEXT527 : BOOL ;	//TEXT N.527
    TEXT528 : BOOL ;	//TEXT N.528
    TEXT513 : BOOL ;	//TEXT N.513
    TEXT514 : BOOL ;	//TEXT N.514
    TEXT515 : BOOL ;	//TEXT N.515
    TEXT516 : BOOL ;	//TEXT N.516
    TEXT517 : BOOL ;	//TEXT N.517
    TEXT518 : BOOL ;	//TEXT N.518
    TEXT519 : BOOL ;	//TEXT N.519
    TEXT520 : BOOL ;	//TEXT N.520
    TEXT537 : BOOL ;	//TEXT N.537
    TEXT538 : BOOL ;	//TEXT N.538
    TEXT539 : BOOL ;	//TEXT N.539
    TEXT540 : BOOL ;	//TEXT N.540
    TEXT541 : BOOL ;	//TEXT N.541
    TEXT542 : BOOL ;	//TEXT N.542
    TEXT543 : BOOL ;	//TEXT N.543
    TEXT544 : BOOL ;	//TEXT N.544
    TEXT529 : BOOL ;	//TEXT N.529
    TEXT530 : BOOL ;	//TEXT N.530
    TEXT531 : BOOL ;	//TEXT N.531
    TEXT532 : BOOL ;	//TEXT N.532
    TEXT533 : BOOL ;	//TEXT N.533
    TEXT534 : BOOL ;	//TEXT N.534
    TEXT535 : BOOL ;	//TEXT N.535
    TEXT536 : BOOL ;	//TEXT N.536
    TEXT553 : BOOL ;	//TEXT N.553
    TEXT554 : BOOL ;	//TEXT N.554
    TEXT555 : BOOL ;	//TEXT N.555
    TEXT556 : BOOL ;	//TEXT N.556
    TEXT557 : BOOL ;	//TEXT N.557
    TEXT558 : BOOL ;	//TEXT N.558
    TEXT559 : BOOL ;	//TEXT N.559
    TEXT560 : BOOL ;	//TEXT N.560
    TEXT545 : BOOL ;	//TEXT N.545
    TEXT546 : BOOL ;	//TEXT N.546
    TEXT547 : BOOL ;	//TEXT N.547
    TEXT548 : BOOL ;	//TEXT N.548
    TEXT549 : BOOL ;	//TEXT N.549
    TEXT550 : BOOL ;	//TEXT N.550
    TEXT551 : BOOL ;	//TEXT N.551
    TEXT552 : BOOL ;	//TEXT N.552
    TEXT569 : BOOL ;	//TEXT N.569
    TEXT570 : BOOL ;	//TEXT N.570
    TEXT571 : BOOL ;	//TEXT N.571
    TEXT572 : BOOL ;	//TEXT N.572
    TEXT573 : BOOL ;	//TEXT N.573
    TEXT574 : BOOL ;	//TEXT N.574
    TEXT575 : BOOL ;	//TEXT N.575
    TEXT576 : BOOL ;	//TEXT N.576
    TEXT561 : BOOL ;	//TEXT N.561
    TEXT562 : BOOL ;	//TEXT N.562
    TEXT563 : BOOL ;	//TEXT N.563
    TEXT564 : BOOL ;	//TEXT N.564
    TEXT565 : BOOL ;	//TEXT N.565
    TEXT566 : BOOL ;	//TEXT N.566
    TEXT567 : BOOL ;	//TEXT N.567
    TEXT568 : BOOL ;	//TEXT N.568
    TEXT585 : BOOL ;	//TEXT N.585
    TEXT586 : BOOL ;	//TEXT N.586
    TEXT587 : BOOL ;	//TEXT N.587
    TEXT588 : BOOL ;	//TEXT N.588
    TEXT589 : BOOL ;	//TEXT N.589
    TEXT590 : BOOL ;	//TEXT N.590
    TEXT591 : BOOL ;	//TEXT N.591
    TEXT592 : BOOL ;	//TEXT N.592
    TEXT577 : BOOL ;	//TEXT N.577
    TEXT578 : BOOL ;	//TEXT N.578
    TEXT579 : BOOL ;	//TEXT N.579
    TEXT580 : BOOL ;	//TEXT N.580
    TEXT581 : BOOL ;	//TEXT N.581
    TEXT582 : BOOL ;	//TEXT N.582
    TEXT583 : BOOL ;	//TEXT N.583
    TEXT584 : BOOL ;	//TEXT N.584
    TEXT601 : BOOL ;	//TEXT N.601
    TEXT602 : BOOL ;	//TEXT N.602
    TEXT603 : BOOL ;	//TEXT N.603
    TEXT604 : BOOL ;	//TEXT N.604
    TEXT605 : BOOL ;	//TEXT N.605
    TEXT606 : BOOL ;	//TEXT N.606
    TEXT607 : BOOL ;	//TEXT N.607
    TEXT608 : BOOL ;	//TEXT N.608
    TEXT593 : BOOL ;	//TEXT N.593
    TEXT594 : BOOL ;	//TEXT N.594
    TEXT595 : BOOL ;	//TEXT N.595
    TEXT596 : BOOL ;	//TEXT N.596
    TEXT597 : BOOL ;	//TEXT N.597
    TEXT598 : BOOL ;	//TEXT N.598
    TEXT599 : BOOL ;	//TEXT N.599
    TEXT600 : BOOL ;	//TEXT N.600
    TEXT617 : BOOL ;	//TEXT N.617
    TEXT618 : BOOL ;	//TEXT N.618
    TEXT619 : BOOL ;	//TEXT N.619
    TEXT620 : BOOL ;	//TEXT N.620
    TEXT621 : BOOL ;	//TEXT N.621
    TEXT622 : BOOL ;	//TEXT N.622
    TEXT623 : BOOL ;	//TEXT N.623
    TEXT624 : BOOL ;	//TEXT N.624
    TEXT609 : BOOL ;	//TEXT N.609
    TEXT610 : BOOL ;	//TEXT N.610
    TEXT611 : BOOL ;	//TEXT N.611
    TEXT612 : BOOL ;	//TEXT N.612
    TEXT613 : BOOL ;	//TEXT N.613
    TEXT614 : BOOL ;	//TEXT N.614
    TEXT615 : BOOL ;	//TEXT N.615
    TEXT616 : BOOL ;	//TEXT N.616
    TEXT633 : BOOL ;	//TEXT N.633
    TEXT634 : BOOL ;	//TEXT N.634
    TEXT635 : BOOL ;	//TEXT N.635
    TEXT636 : BOOL ;	//TEXT N.636
    TEXT637 : BOOL ;	//TEXT N.637
    TEXT638 : BOOL ;	//TEXT N.638
    TEXT639 : BOOL ;	//TEXT N.639
    TEXT640 : BOOL ;	//TEXT N.640
    TEXT625 : BOOL ;	//TEXT N.625
    TEXT626 : BOOL ;	//TEXT N.626
    TEXT627 : BOOL ;	//TEXT N.627
    TEXT628 : BOOL ;	//TEXT N.628
    TEXT629 : BOOL ;	//TEXT N.629
    TEXT630 : BOOL ;	//TEXT N.630
    TEXT631 : BOOL ;	//TEXT N.631
    TEXT632 : BOOL ;	//TEXT N.632
   END_STRUCT ;
   AcquisizioniPLC : STRUCT
    TEXT9 : BOOL ;	//TEXT N.9
    TEXT10 : BOOL ;	//TEXT N.10
    TEXT11 : BOOL ;	//TEXT N.11
    TEXT12 : BOOL ;	//TEXT N.12
    TEXT13 : BOOL ;	//TEXT N.13
    TEXT14 : BOOL ;	//TEXT N.14
    TEXT15 : BOOL ;	//TEXT N.15
    TEXT16 : BOOL ;	//TEXT N.16
    TEXT1 : BOOL ;	//TEXT N.1
    TEXT2 : BOOL ;	//TEXT N.2
    TEXT3 : BOOL ;	//TEXT N.3
    TEXT4 : BOOL ;	//TEXT N.4
    TEXT5 : BOOL ;	//TEXT N.5
    TEXT6 : BOOL ;	//TEXT N.6
    TEXT7 : BOOL ;	//TEXT N.7
    TEXT8 : BOOL ;	//TEXT N.8
    TEXT25 : BOOL ;	//TEXT N.25
    TEXT26 : BOOL ;	//TEXT N.26
    TEXT27 : BOOL ;	//TEXT N.27
    TEXT28 : BOOL ;	//TEXT N.28
    TEXT29 : BOOL ;	//TEXT N.29
    TEXT30 : BOOL ;	//TEXT N.30
    TEXT31 : BOOL ;	//TEXT N.31
    TEXT32 : BOOL ;	//TEXT N.32
    TEXT17 : BOOL ;	//TEXT N.17
    TEXT18 : BOOL ;	//TEXT N.18
    TEXT19 : BOOL ;	//TEXT N.19
    TEXT20 : BOOL ;	//TEXT N.20
    TEXT21 : BOOL ;	//TEXT N.21
    TEXT22 : BOOL ;	//TEXT N.22
    TEXT23 : BOOL ;	//TEXT N.23
    TEXT24 : BOOL ;	//TEXT N.24
    TEXT41 : BOOL ;	//TEXT N.41
    TEXT42 : BOOL ;	//TEXT N.42
    TEXT43 : BOOL ;	//TEXT N.43
    TEXT44 : BOOL ;	//TEXT N.44
    TEXT45 : BOOL ;	//TEXT N.45
    TEXT46 : BOOL ;	//TEXT N.46
    TEXT47 : BOOL ;	//TEXT N.47
    TEXT48 : BOOL ;	//TEXT N.48
    TEXT33 : BOOL ;	//TEXT N.33
    TEXT34 : BOOL ;	//TEXT N.34
    TEXT35 : BOOL ;	//TEXT N.35
    TEXT36 : BOOL ;	//TEXT N.36
    TEXT37 : BOOL ;	//TEXT N.37
    TEXT38 : BOOL ;	//TEXT N.38
    TEXT39 : BOOL ;	//TEXT N.39
    TEXT40 : BOOL ;	//TEXT N.40
    TEXT57 : BOOL ;	//TEXT N.57
    TEXT58 : BOOL ;	//TEXT N.58
    TEXT59 : BOOL ;	//TEXT N.59
    TEXT60 : BOOL ;	//TEXT N.60
    TEXT61 : BOOL ;	//TEXT N.61
    TEXT62 : BOOL ;	//TEXT N.62
    TEXT63 : BOOL ;	//TEXT N.63
    TEXT64 : BOOL ;	//TEXT N.64
    TEXT49 : BOOL ;	//TEXT N.49
    TEXT50 : BOOL ;	//TEXT N.50
    TEXT51 : BOOL ;	//TEXT N.51
    TEXT52 : BOOL ;	//TEXT N.52
    TEXT53 : BOOL ;	//TEXT N.53
    TEXT54 : BOOL ;	//TEXT N.54
    TEXT55 : BOOL ;	//TEXT N.55
    TEXT56 : BOOL ;	//TEXT N.56
    TEXT73 : BOOL ;	//TEXT N.73
    TEXT74 : BOOL ;	//TEXT N.74
    TEXT75 : BOOL ;	//TEXT N.75
    TEXT76 : BOOL ;	//TEXT N.76
    TEXT77 : BOOL ;	//TEXT N.77
    TEXT78 : BOOL ;	//TEXT N.78
    TEXT79 : BOOL ;	//TEXT N.79
    TEXT80 : BOOL ;	//TEXT N.80
    TEXT65 : BOOL ;	//TEXT N.65
    TEXT66 : BOOL ;	//TEXT N.66
    TEXT67 : BOOL ;	//TEXT N.67
    TEXT68 : BOOL ;	//TEXT N.68
    TEXT69 : BOOL ;	//TEXT N.69
    TEXT70 : BOOL ;	//TEXT N.70
    TEXT71 : BOOL ;	//TEXT N.71
    TEXT72 : BOOL ;	//TEXT N.72
    TEXT89 : BOOL ;	//TEXT N.89
    TEXT90 : BOOL ;	//TEXT N.90
    TEXT91 : BOOL ;	//TEXT N.91
    TEXT92 : BOOL ;	//TEXT N.92
    TEXT93 : BOOL ;	//TEXT N.93
    TEXT94 : BOOL ;	//TEXT N.94
    TEXT95 : BOOL ;	//TEXT N.95
    TEXT96 : BOOL ;	//TEXT N.96
    TEXT81 : BOOL ;	//TEXT N.81
    TEXT82 : BOOL ;	//TEXT N.82
    TEXT83 : BOOL ;	//TEXT N.83
    TEXT84 : BOOL ;	//TEXT N.84
    TEXT85 : BOOL ;	//TEXT N.85
    TEXT86 : BOOL ;	//TEXT N.86
    TEXT87 : BOOL ;	//TEXT N.87
    TEXT88 : BOOL ;	//TEXT N.88
    TEXT105 : BOOL ;	//TEXT N.105
    TEXT106 : BOOL ;	//TEXT N.106
    TEXT107 : BOOL ;	//TEXT N.107
    TEXT108 : BOOL ;	//TEXT N.108
    TEXT109 : BOOL ;	//TEXT N.109
    TEXT110 : BOOL ;	//TEXT N.110
    TEXT111 : BOOL ;	//TEXT N.111
    TEXT112 : BOOL ;	//TEXT N.112
    TEXT97 : BOOL ;	//TEXT N.17
    TEXT98 : BOOL ;	//TEXT N.18
    TEXT99 : BOOL ;	//TEXT N.19
    TEXT100 : BOOL ;	//TEXT N.100
    TEXT101 : BOOL ;	//TEXT N.101
    TEXT102 : BOOL ;	//TEXT N.102
    TEXT103 : BOOL ;	//TEXT N.103
    TEXT104 : BOOL ;	//TEXT N.104
    TEXT121 : BOOL ;	//TEXT N.121
    TEXT122 : BOOL ;	//TEXT N.122
    TEXT123 : BOOL ;	//TEXT N.123
    TEXT124 : BOOL ;	//TEXT N.124
    TEXT125 : BOOL ;	//TEXT N.125
    TEXT126 : BOOL ;	//TEXT N.126
    TEXT127 : BOOL ;	//TEXT N.127
    TEXT128 : BOOL ;	//TEXT N.128
    TEXT113 : BOOL ;	//TEXT N.113
    TEXT114 : BOOL ;	//TEXT N.114
    TEXT115 : BOOL ;	//TEXT N.115
    TEXT116 : BOOL ;	//TEXT N.116
    TEXT117 : BOOL ;	//TEXT N.117
    TEXT118 : BOOL ;	//TEXT N.118
    TEXT119 : BOOL ;	//TEXT N.119
    TEXT120 : BOOL ;	//TEXT N.120
    TEXT137 : BOOL ;	//TEXT N.137
    TEXT138 : BOOL ;	//TEXT N.138
    TEXT139 : BOOL ;	//TEXT N.139
    TEXT140 : BOOL ;	//TEXT N.140
    TEXT141 : BOOL ;	//TEXT N.141
    TEXT142 : BOOL ;	//TEXT N.142
    TEXT143 : BOOL ;	//TEXT N.143
    TEXT144 : BOOL ;	//TEXT N.144
    TEXT129 : BOOL ;	//TEXT N.129
    TEXT130 : BOOL ;	//TEXT N.130
    TEXT131 : BOOL ;	//TEXT N.131
    TEXT132 : BOOL ;	//TEXT N.132
    TEXT133 : BOOL ;	//TEXT N.133
    TEXT134 : BOOL ;	//TEXT N.134
    TEXT135 : BOOL ;	//TEXT N.135
    TEXT136 : BOOL ;	//TEXT N.136
    TEXT153 : BOOL ;	//TEXT N.153
    TEXT154 : BOOL ;	//TEXT N.154
    TEXT155 : BOOL ;	//TEXT N.155
    TEXT156 : BOOL ;	//TEXT N.156
    TEXT157 : BOOL ;	//TEXT N.157
    TEXT158 : BOOL ;	//TEXT N.158
    TEXT159 : BOOL ;	//TEXT N.159
    TEXT160 : BOOL ;	//TEXT N.160
    TEXT145 : BOOL ;	//TEXT N.145
    TEXT146 : BOOL ;	//TEXT N.146
    TEXT147 : BOOL ;	//TEXT N.147
    TEXT148 : BOOL ;	//TEXT N.148
    TEXT149 : BOOL ;	//TEXT N.149
    TEXT150 : BOOL ;	//TEXT N.150
    TEXT151 : BOOL ;	//TEXT N.151
    TEXT152 : BOOL ;	//TEXT N.152
    TEXT169 : BOOL ;	//TEXT N.169
    TEXT170 : BOOL ;	//TEXT N.170
    TEXT171 : BOOL ;	//TEXT N.171
    TEXT172 : BOOL ;	//TEXT N.172
    TEXT173 : BOOL ;	//TEXT N.173
    TEXT174 : BOOL ;	//TEXT N.174
    TEXT175 : BOOL ;	//TEXT N.175
    TEXT176 : BOOL ;	//TEXT N.176
    TEXT161 : BOOL ;	//TEXT N.161
    TEXT162 : BOOL ;	//TEXT N.162
    TEXT163 : BOOL ;	//TEXT N.163
    TEXT164 : BOOL ;	//TEXT N.164
    TEXT165 : BOOL ;	//TEXT N.165
    TEXT166 : BOOL ;	//TEXT N.166
    TEXT167 : BOOL ;	//TEXT N.167
    TEXT168 : BOOL ;	//TEXT N.168
    TEXT185 : BOOL ;	//TEXT N.185
    TEXT186 : BOOL ;	//TEXT N.186
    TEXT187 : BOOL ;	//TEXT N.187
    TEXT188 : BOOL ;	//TEXT N.188
    TEXT189 : BOOL ;	//TEXT N.189
    TEXT190 : BOOL ;	//TEXT N.190
    TEXT191 : BOOL ;	//TEXT N.191
    TEXT192 : BOOL ;	//TEXT N.192
    TEXT177 : BOOL ;	//TEXT N.177
    TEXT178 : BOOL ;	//TEXT N.178
    TEXT179 : BOOL ;	//TEXT N.179
    TEXT180 : BOOL ;	//TEXT N.180
    TEXT181 : BOOL ;	//TEXT N.181
    TEXT182 : BOOL ;	//TEXT N.182
    TEXT183 : BOOL ;	//TEXT N.183
    TEXT184 : BOOL ;	//TEXT N.184
    TEXT201 : BOOL ;	//TEXT N.201
    TEXT202 : BOOL ;	//TEXT N.202
    TEXT203 : BOOL ;	//TEXT N.203
    TEXT204 : BOOL ;	//TEXT N.204
    TEXT205 : BOOL ;	//TEXT N.205
    TEXT206 : BOOL ;	//TEXT N.206
    TEXT207 : BOOL ;	//TEXT N.207
    TEXT208 : BOOL ;	//TEXT N.208
    TEXT193 : BOOL ;	//TEXT N.193
    TEXT194 : BOOL ;	//TEXT N.194
    TEXT195 : BOOL ;	//TEXT N.195
    TEXT196 : BOOL ;	//TEXT N.196
    TEXT197 : BOOL ;	//TEXT N.197
    TEXT198 : BOOL ;	//TEXT N.198
    TEXT199 : BOOL ;	//TEXT N.199
    TEXT200 : BOOL ;	//TEXT N.200
    TEXT217 : BOOL ;	//TEXT N.217
    TEXT218 : BOOL ;	//TEXT N.218
    TEXT219 : BOOL ;	//TEXT N.219
    TEXT220 : BOOL ;	//TEXT N.220
    TEXT221 : BOOL ;	//TEXT N.221
    TEXT222 : BOOL ;	//TEXT N.222
    TEXT223 : BOOL ;	//TEXT N.223
    TEXT224 : BOOL ;	//TEXT N.224
    TEXT209 : BOOL ;	//TEXT N.209
    TEXT210 : BOOL ;	//TEXT N.210
    TEXT211 : BOOL ;	//TEXT N.211
    TEXT212 : BOOL ;	//TEXT N.212
    TEXT213 : BOOL ;	//TEXT N.213
    TEXT214 : BOOL ;	//TEXT N.214
    TEXT215 : BOOL ;	//TEXT N.215
    TEXT216 : BOOL ;	//TEXT N.216
    TEXT233 : BOOL ;	//TEXT N.233
    TEXT234 : BOOL ;	//TEXT N.234
    TEXT235 : BOOL ;	//TEXT N.235
    TEXT236 : BOOL ;	//TEXT N.236
    TEXT237 : BOOL ;	//TEXT N.237
    TEXT238 : BOOL ;	//TEXT N.238
    TEXT239 : BOOL ;	//TEXT N.239
    TEXT240 : BOOL ;	//TEXT N.240
    TEXT225 : BOOL ;	//TEXT N.225
    TEXT226 : BOOL ;	//TEXT N.226
    TEXT227 : BOOL ;	//TEXT N.227
    TEXT228 : BOOL ;	//TEXT N.228
    TEXT229 : BOOL ;	//TEXT N.229
    TEXT230 : BOOL ;	//TEXT N.230
    TEXT231 : BOOL ;	//TEXT N.231
    TEXT232 : BOOL ;	//TEXT N.232
    TEXT249 : BOOL ;	//TEXT N.249
    TEXT250 : BOOL ;	//TEXT N.250
    TEXT251 : BOOL ;	//TEXT N.251
    TEXT252 : BOOL ;	//TEXT N.252
    TEXT253 : BOOL ;	//TEXT N.253
    TEXT254 : BOOL ;	//TEXT N.254
    TEXT255 : BOOL ;	//TEXT N.255
    TEXT256 : BOOL ;	//TEXT N.256
    TEXT241 : BOOL ;	//TEXT N.241
    TEXT242 : BOOL ;	//TEXT N.242
    TEXT243 : BOOL ;	//TEXT N.243
    TEXT244 : BOOL ;	//TEXT N.244
    TEXT245 : BOOL ;	//TEXT N.245
    TEXT246 : BOOL ;	//TEXT N.246
    TEXT247 : BOOL ;	//TEXT N.247
    TEXT248 : BOOL ;	//TEXT N.248
    TEXT265 : BOOL ;	//TEXT N.265
    TEXT266 : BOOL ;	//TEXT N.266
    TEXT267 : BOOL ;	//TEXT N.267
    TEXT268 : BOOL ;	//TEXT N.268
    TEXT269 : BOOL ;	//TEXT N.269
    TEXT270 : BOOL ;	//TEXT N.270
    TEXT271 : BOOL ;	//TEXT N.271
    TEXT272 : BOOL ;	//TEXT N.272
    TEXT257 : BOOL ;	//TEXT N.257
    TEXT258 : BOOL ;	//TEXT N.258
    TEXT259 : BOOL ;	//TEXT N.259
    TEXT260 : BOOL ;	//TEXT N.260
    TEXT261 : BOOL ;	//TEXT N.261
    TEXT262 : BOOL ;	//TEXT N.262
    TEXT263 : BOOL ;	//TEXT N.263
    TEXT264 : BOOL ;	//TEXT N.264
    TEXT281 : BOOL ;	//TEXT N.281
    TEXT282 : BOOL ;	//TEXT N.282
    TEXT283 : BOOL ;	//TEXT N.283
    TEXT284 : BOOL ;	//TEXT N.284
    TEXT285 : BOOL ;	//TEXT N.285
    TEXT286 : BOOL ;	//TEXT N.286
    TEXT287 : BOOL ;	//TEXT N.287
    TEXT288 : BOOL ;	//TEXT N.288
    TEXT273 : BOOL ;	//TEXT N.273
    TEXT274 : BOOL ;	//TEXT N.274
    TEXT275 : BOOL ;	//TEXT N.275
    TEXT276 : BOOL ;	//TEXT N.276
    TEXT277 : BOOL ;	//TEXT N.277
    TEXT278 : BOOL ;	//TEXT N.278
    TEXT279 : BOOL ;	//TEXT N.279
    TEXT280 : BOOL ;	//TEXT N.280
    TEXT297 : BOOL ;	//TEXT N.297
    TEXT298 : BOOL ;	//TEXT N.298
    TEXT299 : BOOL ;	//TEXT N.299
    TEXT300 : BOOL ;	//TEXT N.300
    TEXT301 : BOOL ;	//TEXT N.301
    TEXT302 : BOOL ;	//TEXT N.302
    TEXT303 : BOOL ;	//TEXT N.303
    TEXT304 : BOOL ;	//TEXT N.304
    TEXT289 : BOOL ;	//TEXT N.289
    TEXT290 : BOOL ;	//TEXT N.290
    TEXT291 : BOOL ;	//TEXT N.291
    TEXT292 : BOOL ;	//TEXT N.292
    TEXT293 : BOOL ;	//TEXT N.293
    TEXT294 : BOOL ;	//TEXT N.294
    TEXT295 : BOOL ;	//TEXT N.295
    TEXT296 : BOOL ;	//TEXT N.296
    TEXT313 : BOOL ;	//TEXT N.313
    TEXT314 : BOOL ;	//TEXT N.314
    TEXT315 : BOOL ;	//TEXT N.315
    TEXT316 : BOOL ;	//TEXT N.316
    TEXT317 : BOOL ;	//TEXT N.317
    TEXT318 : BOOL ;	//TEXT N.318
    TEXT319 : BOOL ;	//TEXT N.319
    TEXT320 : BOOL ;	//TEXT N.320
    TEXT305 : BOOL ;	//TEXT N.305
    TEXT306 : BOOL ;	//TEXT N.306
    TEXT307 : BOOL ;	//TEXT N.307
    TEXT308 : BOOL ;	//TEXT N.308
    TEXT309 : BOOL ;	//TEXT N.309
    TEXT310 : BOOL ;	//TEXT N.310
    TEXT311 : BOOL ;	//TEXT N.311
    TEXT312 : BOOL ;	//TEXT N.312
    TEXT329 : BOOL ;	//TEXT N.329
    TEXT330 : BOOL ;	//TEXT N.330
    TEXT331 : BOOL ;	//TEXT N.331
    TEXT332 : BOOL ;	//TEXT N.332
    TEXT333 : BOOL ;	//TEXT N.333
    TEXT334 : BOOL ;	//TEXT N.334
    TEXT335 : BOOL ;	//TEXT N.335
    TEXT336 : BOOL ;	//TEXT N.336
    TEXT321 : BOOL ;	//TEXT N.321
    TEXT322 : BOOL ;	//TEXT N.322
    TEXT323 : BOOL ;	//TEXT N.323
    TEXT324 : BOOL ;	//TEXT N.324
    TEXT325 : BOOL ;	//TEXT N.325
    TEXT326 : BOOL ;	//TEXT N.326
    TEXT327 : BOOL ;	//TEXT N.327
    TEXT328 : BOOL ;	//TEXT N.328
    TEXT345 : BOOL ;	//TEXT N.345
    TEXT346 : BOOL ;	//TEXT N.346
    TEXT347 : BOOL ;	//TEXT N.347
    TEXT348 : BOOL ;	//TEXT N.348
    TEXT349 : BOOL ;	//TEXT N.349
    TEXT350 : BOOL ;	//TEXT N.350
    TEXT351 : BOOL ;	//TEXT N.351
    TEXT352 : BOOL ;	//TEXT N.352
    TEXT337 : BOOL ;	//TEXT N.337
    TEXT338 : BOOL ;	//TEXT N.338
    TEXT339 : BOOL ;	//TEXT N.339
    TEXT340 : BOOL ;	//TEXT N.340
    TEXT341 : BOOL ;	//TEXT N.341
    TEXT342 : BOOL ;	//TEXT N.342
    TEXT343 : BOOL ;	//TEXT N.343
    TEXT344 : BOOL ;	//TEXT N.344
    TEXT361 : BOOL ;	//TEXT N.361
    TEXT362 : BOOL ;	//TEXT N.362
    TEXT363 : BOOL ;	//TEXT N.363
    TEXT364 : BOOL ;	//TEXT N.364
    TEXT365 : BOOL ;	//TEXT N.365
    TEXT366 : BOOL ;	//TEXT N.366
    TEXT367 : BOOL ;	//TEXT N.367
    TEXT368 : BOOL ;	//TEXT N.368
    TEXT353 : BOOL ;	//TEXT N.353
    TEXT354 : BOOL ;	//TEXT N.354
    TEXT355 : BOOL ;	//TEXT N.355
    TEXT356 : BOOL ;	//TEXT N.356
    TEXT357 : BOOL ;	//TEXT N.357
    TEXT358 : BOOL ;	//TEXT N.358
    TEXT359 : BOOL ;	//TEXT N.359
    TEXT360 : BOOL ;	//TEXT N.360
    TEXT377 : BOOL ;	//TEXT N.377
    TEXT378 : BOOL ;	//TEXT N.378
    TEXT379 : BOOL ;	//TEXT N.379
    TEXT380 : BOOL ;	//TEXT N.380
    TEXT381 : BOOL ;	//TEXT N.381
    TEXT382 : BOOL ;	//TEXT N.382
    TEXT383 : BOOL ;	//TEXT N.383
    TEXT384 : BOOL ;	//TEXT N.384
    TEXT369 : BOOL ;	//TEXT N.369
    TEXT370 : BOOL ;	//TEXT N.370
    TEXT371 : BOOL ;	//TEXT N.371
    TEXT372 : BOOL ;	//TEXT N.372
    TEXT373 : BOOL ;	//TEXT N.373
    TEXT374 : BOOL ;	//TEXT N.374
    TEXT375 : BOOL ;	//TEXT N.375
    TEXT376 : BOOL ;	//TEXT N.376
    TEXT393 : BOOL ;	//TEXT N.393
    TEXT394 : BOOL ;	//TEXT N.394
    TEXT395 : BOOL ;	//TEXT N.395
    TEXT396 : BOOL ;	//TEXT N.396
    TEXT397 : BOOL ;	//TEXT N.397
    TEXT398 : BOOL ;	//TEXT N.398
    TEXT399 : BOOL ;	//TEXT N.399
    TEXT400 : BOOL ;	//TEXT N.400
    TEXT385 : BOOL ;	//TEXT N.385
    TEXT386 : BOOL ;	//TEXT N.386
    TEXT387 : BOOL ;	//TEXT N.387
    TEXT388 : BOOL ;	//TEXT N.388
    TEXT389 : BOOL ;	//TEXT N.389
    TEXT390 : BOOL ;	//TEXT N.390
    TEXT391 : BOOL ;	//TEXT N.391
    TEXT392 : BOOL ;	//TEXT N.392
    TEXT409 : BOOL ;	//TEXT N.409
    TEXT410 : BOOL ;	//TEXT N.410
    TEXT411 : BOOL ;	//TEXT N.411
    TEXT412 : BOOL ;	//TEXT N.412
    TEXT413 : BOOL ;	//TEXT N.413
    TEXT414 : BOOL ;	//TEXT N.414
    TEXT415 : BOOL ;	//TEXT N.415
    TEXT416 : BOOL ;	//TEXT N.416
    TEXT401 : BOOL ;	//TEXT N.401
    TEXT402 : BOOL ;	//TEXT N.402
    TEXT403 : BOOL ;	//TEXT N.403
    TEXT404 : BOOL ;	//TEXT N.404
    TEXT405 : BOOL ;	//TEXT N.405
    TEXT406 : BOOL ;	//TEXT N.406
    TEXT407 : BOOL ;	//TEXT N.407
    TEXT408 : BOOL ;	//TEXT N.408
    TEXT425 : BOOL ;	//TEXT N.425
    TEXT426 : BOOL ;	//TEXT N.426
    TEXT427 : BOOL ;	//TEXT N.427
    TEXT428 : BOOL ;	//TEXT N.428
    TEXT429 : BOOL ;	//TEXT N.429
    TEXT430 : BOOL ;	//TEXT N.430
    TEXT431 : BOOL ;	//TEXT N.431
    TEXT432 : BOOL ;	//TEXT N.432
    TEXT417 : BOOL ;	//TEXT N.417
    TEXT418 : BOOL ;	//TEXT N.418
    TEXT419 : BOOL ;	//TEXT N.419
    TEXT420 : BOOL ;	//TEXT N.420
    TEXT421 : BOOL ;	//TEXT N.421
    TEXT422 : BOOL ;	//TEXT N.422
    TEXT423 : BOOL ;	//TEXT N.423
    TEXT424 : BOOL ;	//TEXT N.424
    TEXT441 : BOOL ;	//TEXT N.441
    TEXT442 : BOOL ;	//TEXT N.442
    TEXT443 : BOOL ;	//TEXT N.443
    TEXT444 : BOOL ;	//TEXT N.444
    TEXT445 : BOOL ;	//TEXT N.445
    TEXT446 : BOOL ;	//TEXT N.446
    TEXT447 : BOOL ;	//TEXT N.447
    TEXT448 : BOOL ;	//TEXT N.448
    TEXT433 : BOOL ;	//TEXT N.433
    TEXT434 : BOOL ;	//TEXT N.434
    TEXT435 : BOOL ;	//TEXT N.435
    TEXT436 : BOOL ;	//TEXT N.436
    TEXT437 : BOOL ;	//TEXT N.437
    TEXT438 : BOOL ;	//TEXT N.438
    TEXT439 : BOOL ;	//TEXT N.439
    TEXT440 : BOOL ;	//TEXT N.440
    TEXT457 : BOOL ;	//TEXT N.457
    TEXT458 : BOOL ;	//TEXT N.458
    TEXT459 : BOOL ;	//TEXT N.459
    TEXT460 : BOOL ;	//TEXT N.460
    TEXT461 : BOOL ;	//TEXT N.461
    TEXT462 : BOOL ;	//TEXT N.462
    TEXT463 : BOOL ;	//TEXT N.463
    TEXT464 : BOOL ;	//TEXT N.464
    TEXT449 : BOOL ;	//TEXT N.449
    TEXT450 : BOOL ;	//TEXT N.450
    TEXT451 : BOOL ;	//TEXT N.451
    TEXT452 : BOOL ;	//TEXT N.452
    TEXT453 : BOOL ;	//TEXT N.453
    TEXT454 : BOOL ;	//TEXT N.454
    TEXT455 : BOOL ;	//TEXT N.455
    TEXT456 : BOOL ;	//TEXT N.456
    TEXT473 : BOOL ;	//TEXT N.473
    TEXT474 : BOOL ;	//TEXT N.474
    TEXT475 : BOOL ;	//TEXT N.475
    TEXT476 : BOOL ;	//TEXT N.476
    TEXT477 : BOOL ;	//TEXT N.477
    TEXT478 : BOOL ;	//TEXT N.478
    TEXT479 : BOOL ;	//TEXT N.479
    TEXT480 : BOOL ;	//TEXT N.480
    TEXT465 : BOOL ;	//TEXT N.465
    TEXT466 : BOOL ;	//TEXT N.466
    TEXT467 : BOOL ;	//TEXT N.467
    TEXT468 : BOOL ;	//TEXT N.468
    TEXT469 : BOOL ;	//TEXT N.469
    TEXT470 : BOOL ;	//TEXT N.470
    TEXT471 : BOOL ;	//TEXT N.471
    TEXT472 : BOOL ;	//TEXT N.472
    TEXT489 : BOOL ;	//TEXT N.489
    TEXT490 : BOOL ;	//TEXT N.490
    TEXT491 : BOOL ;	//TEXT N.491
    TEXT492 : BOOL ;	//TEXT N.492
    TEXT493 : BOOL ;	//TEXT N.493
    TEXT494 : BOOL ;	//TEXT N.494
    TEXT495 : BOOL ;	//TEXT N.495
    TEXT496 : BOOL ;	//TEXT N.496
    TEXT481 : BOOL ;	//TEXT N.481
    TEXT482 : BOOL ;	//TEXT N.482
    TEXT483 : BOOL ;	//TEXT N.483
    TEXT484 : BOOL ;	//TEXT N.484
    TEXT485 : BOOL ;	//TEXT N.485
    TEXT486 : BOOL ;	//TEXT N.486
    TEXT487 : BOOL ;	//TEXT N.487
    TEXT488 : BOOL ;	//TEXT N.488
    TEXT505 : BOOL ;	//TEXT N.505
    TEXT506 : BOOL ;	//TEXT N.506
    TEXT507 : BOOL ;	//TEXT N.507
    TEXT508 : BOOL ;	//TEXT N.508
    TEXT509 : BOOL ;	//TEXT N.509
    TEXT510 : BOOL ;	//TEXT N.510
    TEXT511 : BOOL ;	//TEXT N.511
    TEXT512 : BOOL ;	//TEXT N.512
    TEXT497 : BOOL ;	//TEXT N.497
    TEXT498 : BOOL ;	//TEXT N.498
    TEXT499 : BOOL ;	//TEXT N.499
    TEXT500 : BOOL ;	//TEXT N.500
    TEXT501 : BOOL ;	//TEXT N.501
    TEXT502 : BOOL ;	//TEXT N.502
    TEXT503 : BOOL ;	//TEXT N.503
    TEXT504 : BOOL ;	//TEXT N.504
    TEXT521 : BOOL ;	//TEXT N.521
    TEXT522 : BOOL ;	//TEXT N.522
    TEXT523 : BOOL ;	//TEXT N.523
    TEXT524 : BOOL ;	//TEXT N.524
    TEXT525 : BOOL ;	//TEXT N.525
    TEXT526 : BOOL ;	//TEXT N.526
    TEXT527 : BOOL ;	//TEXT N.527
    TEXT528 : BOOL ;	//TEXT N.528
    TEXT513 : BOOL ;	//TEXT N.513
    TEXT514 : BOOL ;	//TEXT N.514
    TEXT515 : BOOL ;	//TEXT N.515
    TEXT516 : BOOL ;	//TEXT N.516
    TEXT517 : BOOL ;	//TEXT N.517
    TEXT518 : BOOL ;	//TEXT N.518
    TEXT519 : BOOL ;	//TEXT N.519
    TEXT520 : BOOL ;	//TEXT N.520
    TEXT537 : BOOL ;	//TEXT N.537
    TEXT538 : BOOL ;	//TEXT N.538
    TEXT539 : BOOL ;	//TEXT N.539
    TEXT540 : BOOL ;	//TEXT N.540
    TEXT541 : BOOL ;	//TEXT N.541
    TEXT542 : BOOL ;	//TEXT N.542
    TEXT543 : BOOL ;	//TEXT N.543
    TEXT544 : BOOL ;	//TEXT N.544
    TEXT529 : BOOL ;	//TEXT N.529
    TEXT530 : BOOL ;	//TEXT N.530
    TEXT531 : BOOL ;	//TEXT N.531
    TEXT532 : BOOL ;	//TEXT N.532
    TEXT533 : BOOL ;	//TEXT N.533
    TEXT534 : BOOL ;	//TEXT N.534
    TEXT535 : BOOL ;	//TEXT N.535
    TEXT536 : BOOL ;	//TEXT N.536
    TEXT553 : BOOL ;	//TEXT N.553
    TEXT554 : BOOL ;	//TEXT N.554
    TEXT555 : BOOL ;	//TEXT N.555
    TEXT556 : BOOL ;	//TEXT N.556
    TEXT557 : BOOL ;	//TEXT N.557
    TEXT558 : BOOL ;	//TEXT N.558
    TEXT559 : BOOL ;	//TEXT N.559
    TEXT560 : BOOL ;	//TEXT N.560
    TEXT545 : BOOL ;	//TEXT N.545
    TEXT546 : BOOL ;	//TEXT N.546
    TEXT547 : BOOL ;	//TEXT N.547
    TEXT548 : BOOL ;	//TEXT N.548
    TEXT549 : BOOL ;	//TEXT N.549
    TEXT550 : BOOL ;	//TEXT N.550
    TEXT551 : BOOL ;	//TEXT N.551
    TEXT552 : BOOL ;	//TEXT N.552
    TEXT569 : BOOL ;	//TEXT N.569
    TEXT570 : BOOL ;	//TEXT N.570
    TEXT571 : BOOL ;	//TEXT N.571
    TEXT572 : BOOL ;	//TEXT N.572
    TEXT573 : BOOL ;	//TEXT N.573
    TEXT574 : BOOL ;	//TEXT N.574
    TEXT575 : BOOL ;	//TEXT N.575
    TEXT576 : BOOL ;	//TEXT N.576
    TEXT561 : BOOL ;	//TEXT N.561
    TEXT562 : BOOL ;	//TEXT N.562
    TEXT563 : BOOL ;	//TEXT N.563
    TEXT564 : BOOL ;	//TEXT N.564
    TEXT565 : BOOL ;	//TEXT N.565
    TEXT566 : BOOL ;	//TEXT N.566
    TEXT567 : BOOL ;	//TEXT N.567
    TEXT568 : BOOL ;	//TEXT N.568
    TEXT585 : BOOL ;	//TEXT N.585
    TEXT586 : BOOL ;	//TEXT N.586
    TEXT587 : BOOL ;	//TEXT N.587
    TEXT588 : BOOL ;	//TEXT N.588
    TEXT589 : BOOL ;	//TEXT N.589
    TEXT590 : BOOL ;	//TEXT N.590
    TEXT591 : BOOL ;	//TEXT N.591
    TEXT592 : BOOL ;	//TEXT N.592
    TEXT577 : BOOL ;	//TEXT N.577
    TEXT578 : BOOL ;	//TEXT N.578
    TEXT579 : BOOL ;	//TEXT N.579
    TEXT580 : BOOL ;	//TEXT N.580
    TEXT581 : BOOL ;	//TEXT N.581
    TEXT582 : BOOL ;	//TEXT N.582
    TEXT583 : BOOL ;	//TEXT N.583
    TEXT584 : BOOL ;	//TEXT N.584
    TEXT601 : BOOL ;	//TEXT N.601
    TEXT602 : BOOL ;	//TEXT N.602
    TEXT603 : BOOL ;	//TEXT N.603
    TEXT604 : BOOL ;	//TEXT N.604
    TEXT605 : BOOL ;	//TEXT N.605
    TEXT606 : BOOL ;	//TEXT N.606
    TEXT607 : BOOL ;	//TEXT N.607
    TEXT608 : BOOL ;	//TEXT N.608
    TEXT593 : BOOL ;	//TEXT N.593
    TEXT594 : BOOL ;	//TEXT N.594
    TEXT595 : BOOL ;	//TEXT N.595
    TEXT596 : BOOL ;	//TEXT N.596
    TEXT597 : BOOL ;	//TEXT N.597
    TEXT598 : BOOL ;	//TEXT N.598
    TEXT599 : BOOL ;	//TEXT N.599
    TEXT600 : BOOL ;	//TEXT N.600
    TEXT617 : BOOL ;	//TEXT N.617
    TEXT618 : BOOL ;	//TEXT N.618
    TEXT619 : BOOL ;	//TEXT N.619
    TEXT620 : BOOL ;	//TEXT N.620
    TEXT621 : BOOL ;	//TEXT N.621
    TEXT622 : BOOL ;	//TEXT N.622
    TEXT623 : BOOL ;	//TEXT N.623
    TEXT624 : BOOL ;	//TEXT N.624
    TEXT609 : BOOL ;	//TEXT N.609
    TEXT610 : BOOL ;	//TEXT N.610
    TEXT611 : BOOL ;	//TEXT N.611
    TEXT612 : BOOL ;	//TEXT N.612
    TEXT613 : BOOL ;	//TEXT N.613
    TEXT614 : BOOL ;	//TEXT N.614
    TEXT615 : BOOL ;	//TEXT N.615
    TEXT616 : BOOL ;	//TEXT N.616
    TEXT633 : BOOL ;	//TEXT N.633
    TEXT634 : BOOL ;	//TEXT N.634
    TEXT635 : BOOL ;	//TEXT N.635
    TEXT636 : BOOL ;	//TEXT N.636
    TEXT637 : BOOL ;	//TEXT N.637
    TEXT638 : BOOL ;	//TEXT N.638
    TEXT639 : BOOL ;	//TEXT N.639
    TEXT640 : BOOL ;	//TEXT N.640
    TEXT625 : BOOL ;	//TEXT N.625
    TEXT626 : BOOL ;	//TEXT N.626
    TEXT627 : BOOL ;	//TEXT N.627
    TEXT628 : BOOL ;	//TEXT N.628
    TEXT629 : BOOL ;	//TEXT N.629
    TEXT630 : BOOL ;	//TEXT N.630
    TEXT631 : BOOL ;	//TEXT N.631
    TEXT632 : BOOL ;	//TEXT N.632
   END_STRUCT ;
   AcquisizioniOP : STRUCT
    TEXT9 : BOOL ;	//TEXT N.9
    TEXT10 : BOOL ;	//TEXT N.10
    TEXT11 : BOOL ;	//TEXT N.11
    TEXT12 : BOOL ;	//TEXT N.12
    TEXT13 : BOOL ;	//TEXT N.13
    TEXT14 : BOOL ;	//TEXT N.14
    TEXT15 : BOOL ;	//TEXT N.15
    TEXT16 : BOOL ;	//TEXT N.16
    TEXT1 : BOOL ;	//TEXT N.1
    TEXT2 : BOOL ;	//TEXT N.2
    TEXT3 : BOOL ;	//TEXT N.3
    TEXT4 : BOOL ;	//TEXT N.4
    TEXT5 : BOOL ;	//TEXT N.5
    TEXT6 : BOOL ;	//TEXT N.6
    TEXT7 : BOOL ;	//TEXT N.7
    TEXT8 : BOOL ;	//TEXT N.8
    TEXT25 : BOOL ;	//TEXT N.25
    TEXT26 : BOOL ;	//TEXT N.26
    TEXT27 : BOOL ;	//TEXT N.27
    TEXT28 : BOOL ;	//TEXT N.28
    TEXT29 : BOOL ;	//TEXT N.29
    TEXT30 : BOOL ;	//TEXT N.30
    TEXT31 : BOOL ;	//TEXT N.31
    TEXT32 : BOOL ;	//TEXT N.32
    TEXT17 : BOOL ;	//TEXT N.17
    TEXT18 : BOOL ;	//TEXT N.18
    TEXT19 : BOOL ;	//TEXT N.19
    TEXT20 : BOOL ;	//TEXT N.20
    TEXT21 : BOOL ;	//TEXT N.21
    TEXT22 : BOOL ;	//TEXT N.22
    TEXT23 : BOOL ;	//TEXT N.23
    TEXT24 : BOOL ;	//TEXT N.24
    TEXT41 : BOOL ;	//TEXT N.41
    TEXT42 : BOOL ;	//TEXT N.42
    TEXT43 : BOOL ;	//TEXT N.43
    TEXT44 : BOOL ;	//TEXT N.44
    TEXT45 : BOOL ;	//TEXT N.45
    TEXT46 : BOOL ;	//TEXT N.46
    TEXT47 : BOOL ;	//TEXT N.47
    TEXT48 : BOOL ;	//TEXT N.48
    TEXT33 : BOOL ;	//TEXT N.33
    TEXT34 : BOOL ;	//TEXT N.34
    TEXT35 : BOOL ;	//TEXT N.35
    TEXT36 : BOOL ;	//TEXT N.36
    TEXT37 : BOOL ;	//TEXT N.37
    TEXT38 : BOOL ;	//TEXT N.38
    TEXT39 : BOOL ;	//TEXT N.39
    TEXT40 : BOOL ;	//TEXT N.40
    TEXT57 : BOOL ;	//TEXT N.57
    TEXT58 : BOOL ;	//TEXT N.58
    TEXT59 : BOOL ;	//TEXT N.59
    TEXT60 : BOOL ;	//TEXT N.60
    TEXT61 : BOOL ;	//TEXT N.61
    TEXT62 : BOOL ;	//TEXT N.62
    TEXT63 : BOOL ;	//TEXT N.63
    TEXT64 : BOOL ;	//TEXT N.64
    TEXT49 : BOOL ;	//TEXT N.49
    TEXT50 : BOOL ;	//TEXT N.50
    TEXT51 : BOOL ;	//TEXT N.51
    TEXT52 : BOOL ;	//TEXT N.52
    TEXT53 : BOOL ;	//TEXT N.53
    TEXT54 : BOOL ;	//TEXT N.54
    TEXT55 : BOOL ;	//TEXT N.55
    TEXT56 : BOOL ;	//TEXT N.56
    TEXT73 : BOOL ;	//TEXT N.73
    TEXT74 : BOOL ;	//TEXT N.74
    TEXT75 : BOOL ;	//TEXT N.75
    TEXT76 : BOOL ;	//TEXT N.76
    TEXT77 : BOOL ;	//TEXT N.77
    TEXT78 : BOOL ;	//TEXT N.78
    TEXT79 : BOOL ;	//TEXT N.79
    TEXT80 : BOOL ;	//TEXT N.80
    TEXT65 : BOOL ;	//TEXT N.65
    TEXT66 : BOOL ;	//TEXT N.66
    TEXT67 : BOOL ;	//TEXT N.67
    TEXT68 : BOOL ;	//TEXT N.68
    TEXT69 : BOOL ;	//TEXT N.69
    TEXT70 : BOOL ;	//TEXT N.70
    TEXT71 : BOOL ;	//TEXT N.71
    TEXT72 : BOOL ;	//TEXT N.72
    TEXT89 : BOOL ;	//TEXT N.89
    TEXT90 : BOOL ;	//TEXT N.90
    TEXT91 : BOOL ;	//TEXT N.91
    TEXT92 : BOOL ;	//TEXT N.92
    TEXT93 : BOOL ;	//TEXT N.93
    TEXT94 : BOOL ;	//TEXT N.94
    TEXT95 : BOOL ;	//TEXT N.95
    TEXT96 : BOOL ;	//TEXT N.96
    TEXT81 : BOOL ;	//TEXT N.81
    TEXT82 : BOOL ;	//TEXT N.82
    TEXT83 : BOOL ;	//TEXT N.83
    TEXT84 : BOOL ;	//TEXT N.84
    TEXT85 : BOOL ;	//TEXT N.85
    TEXT86 : BOOL ;	//TEXT N.86
    TEXT87 : BOOL ;	//TEXT N.87
    TEXT88 : BOOL ;	//TEXT N.88
    TEXT105 : BOOL ;	//TEXT N.105
    TEXT106 : BOOL ;	//TEXT N.106
    TEXT107 : BOOL ;	//TEXT N.107
    TEXT108 : BOOL ;	//TEXT N.108
    TEXT109 : BOOL ;	//TEXT N.109
    TEXT110 : BOOL ;	//TEXT N.110
    TEXT111 : BOOL ;	//TEXT N.111
    TEXT112 : BOOL ;	//TEXT N.112
    TEXT97 : BOOL ;	//TEXT N.17
    TEXT98 : BOOL ;	//TEXT N.18
    TEXT99 : BOOL ;	//TEXT N.19
    TEXT100 : BOOL ;	//TEXT N.100
    TEXT101 : BOOL ;	//TEXT N.101
    TEXT102 : BOOL ;	//TEXT N.102
    TEXT103 : BOOL ;	//TEXT N.103
    TEXT104 : BOOL ;	//TEXT N.104
    TEXT121 : BOOL ;	//TEXT N.121
    TEXT122 : BOOL ;	//TEXT N.122
    TEXT123 : BOOL ;	//TEXT N.123
    TEXT124 : BOOL ;	//TEXT N.124
    TEXT125 : BOOL ;	//TEXT N.125
    TEXT126 : BOOL ;	//TEXT N.126
    TEXT127 : BOOL ;	//TEXT N.127
    TEXT128 : BOOL ;	//TEXT N.128
    TEXT113 : BOOL ;	//TEXT N.113
    TEXT114 : BOOL ;	//TEXT N.114
    TEXT115 : BOOL ;	//TEXT N.115
    TEXT116 : BOOL ;	//TEXT N.116
    TEXT117 : BOOL ;	//TEXT N.117
    TEXT118 : BOOL ;	//TEXT N.118
    TEXT119 : BOOL ;	//TEXT N.119
    TEXT120 : BOOL ;	//TEXT N.120
    TEXT137 : BOOL ;	//TEXT N.137
    TEXT138 : BOOL ;	//TEXT N.138
    TEXT139 : BOOL ;	//TEXT N.139
    TEXT140 : BOOL ;	//TEXT N.140
    TEXT141 : BOOL ;	//TEXT N.141
    TEXT142 : BOOL ;	//TEXT N.142
    TEXT143 : BOOL ;	//TEXT N.143
    TEXT144 : BOOL ;	//TEXT N.144
    TEXT129 : BOOL ;	//TEXT N.129
    TEXT130 : BOOL ;	//TEXT N.130
    TEXT131 : BOOL ;	//TEXT N.131
    TEXT132 : BOOL ;	//TEXT N.132
    TEXT133 : BOOL ;	//TEXT N.133
    TEXT134 : BOOL ;	//TEXT N.134
    TEXT135 : BOOL ;	//TEXT N.135
    TEXT136 : BOOL ;	//TEXT N.136
    TEXT153 : BOOL ;	//TEXT N.153
    TEXT154 : BOOL ;	//TEXT N.154
    TEXT155 : BOOL ;	//TEXT N.155
    TEXT156 : BOOL ;	//TEXT N.156
    TEXT157 : BOOL ;	//TEXT N.157
    TEXT158 : BOOL ;	//TEXT N.158
    TEXT159 : BOOL ;	//TEXT N.159
    TEXT160 : BOOL ;	//TEXT N.160
    TEXT145 : BOOL ;	//TEXT N.145
    TEXT146 : BOOL ;	//TEXT N.146
    TEXT147 : BOOL ;	//TEXT N.147
    TEXT148 : BOOL ;	//TEXT N.148
    TEXT149 : BOOL ;	//TEXT N.149
    TEXT150 : BOOL ;	//TEXT N.150
    TEXT151 : BOOL ;	//TEXT N.151
    TEXT152 : BOOL ;	//TEXT N.152
    TEXT169 : BOOL ;	//TEXT N.169
    TEXT170 : BOOL ;	//TEXT N.170
    TEXT171 : BOOL ;	//TEXT N.171
    TEXT172 : BOOL ;	//TEXT N.172
    TEXT173 : BOOL ;	//TEXT N.173
    TEXT174 : BOOL ;	//TEXT N.174
    TEXT175 : BOOL ;	//TEXT N.175
    TEXT176 : BOOL ;	//TEXT N.176
    TEXT161 : BOOL ;	//TEXT N.161
    TEXT162 : BOOL ;	//TEXT N.162
    TEXT163 : BOOL ;	//TEXT N.163
    TEXT164 : BOOL ;	//TEXT N.164
    TEXT165 : BOOL ;	//TEXT N.165
    TEXT166 : BOOL ;	//TEXT N.166
    TEXT167 : BOOL ;	//TEXT N.167
    TEXT168 : BOOL ;	//TEXT N.168
    TEXT185 : BOOL ;	//TEXT N.185
    TEXT186 : BOOL ;	//TEXT N.186
    TEXT187 : BOOL ;	//TEXT N.187
    TEXT188 : BOOL ;	//TEXT N.188
    TEXT189 : BOOL ;	//TEXT N.189
    TEXT190 : BOOL ;	//TEXT N.190
    TEXT191 : BOOL ;	//TEXT N.191
    TEXT192 : BOOL ;	//TEXT N.192
    TEXT177 : BOOL ;	//TEXT N.177
    TEXT178 : BOOL ;	//TEXT N.178
    TEXT179 : BOOL ;	//TEXT N.179
    TEXT180 : BOOL ;	//TEXT N.180
    TEXT181 : BOOL ;	//TEXT N.181
    TEXT182 : BOOL ;	//TEXT N.182
    TEXT183 : BOOL ;	//TEXT N.183
    TEXT184 : BOOL ;	//TEXT N.184
    TEXT201 : BOOL ;	//TEXT N.201
    TEXT202 : BOOL ;	//TEXT N.202
    TEXT203 : BOOL ;	//TEXT N.203
    TEXT204 : BOOL ;	//TEXT N.204
    TEXT205 : BOOL ;	//TEXT N.205
    TEXT206 : BOOL ;	//TEXT N.206
    TEXT207 : BOOL ;	//TEXT N.207
    TEXT208 : BOOL ;	//TEXT N.208
    TEXT193 : BOOL ;	//TEXT N.193
    TEXT194 : BOOL ;	//TEXT N.194
    TEXT195 : BOOL ;	//TEXT N.195
    TEXT196 : BOOL ;	//TEXT N.196
    TEXT197 : BOOL ;	//TEXT N.197
    TEXT198 : BOOL ;	//TEXT N.198
    TEXT199 : BOOL ;	//TEXT N.199
    TEXT200 : BOOL ;	//TEXT N.200
    TEXT217 : BOOL ;	//TEXT N.217
    TEXT218 : BOOL ;	//TEXT N.218
    TEXT219 : BOOL ;	//TEXT N.219
    TEXT220 : BOOL ;	//TEXT N.220
    TEXT221 : BOOL ;	//TEXT N.221
    TEXT222 : BOOL ;	//TEXT N.222
    TEXT223 : BOOL ;	//TEXT N.223
    TEXT224 : BOOL ;	//TEXT N.224
    TEXT209 : BOOL ;	//TEXT N.209
    TEXT210 : BOOL ;	//TEXT N.210
    TEXT211 : BOOL ;	//TEXT N.211
    TEXT212 : BOOL ;	//TEXT N.212
    TEXT213 : BOOL ;	//TEXT N.213
    TEXT214 : BOOL ;	//TEXT N.214
    TEXT215 : BOOL ;	//TEXT N.215
    TEXT216 : BOOL ;	//TEXT N.216
    TEXT233 : BOOL ;	//TEXT N.233
    TEXT234 : BOOL ;	//TEXT N.234
    TEXT235 : BOOL ;	//TEXT N.235
    TEXT236 : BOOL ;	//TEXT N.236
    TEXT237 : BOOL ;	//TEXT N.237
    TEXT238 : BOOL ;	//TEXT N.238
    TEXT239 : BOOL ;	//TEXT N.239
    TEXT240 : BOOL ;	//TEXT N.240
    TEXT225 : BOOL ;	//TEXT N.225
    TEXT226 : BOOL ;	//TEXT N.226
    TEXT227 : BOOL ;	//TEXT N.227
    TEXT228 : BOOL ;	//TEXT N.228
    TEXT229 : BOOL ;	//TEXT N.229
    TEXT230 : BOOL ;	//TEXT N.230
    TEXT231 : BOOL ;	//TEXT N.231
    TEXT232 : BOOL ;	//TEXT N.232
    TEXT249 : BOOL ;	//TEXT N.249
    TEXT250 : BOOL ;	//TEXT N.250
    TEXT251 : BOOL ;	//TEXT N.251
    TEXT252 : BOOL ;	//TEXT N.252
    TEXT253 : BOOL ;	//TEXT N.253
    TEXT254 : BOOL ;	//TEXT N.254
    TEXT255 : BOOL ;	//TEXT N.255
    TEXT256 : BOOL ;	//TEXT N.256
    TEXT241 : BOOL ;	//TEXT N.241
    TEXT242 : BOOL ;	//TEXT N.242
    TEXT243 : BOOL ;	//TEXT N.243
    TEXT244 : BOOL ;	//TEXT N.244
    TEXT245 : BOOL ;	//TEXT N.245
    TEXT246 : BOOL ;	//TEXT N.246
    TEXT247 : BOOL ;	//TEXT N.247
    TEXT248 : BOOL ;	//TEXT N.248
    TEXT265 : BOOL ;	//TEXT N.265
    TEXT266 : BOOL ;	//TEXT N.266
    TEXT267 : BOOL ;	//TEXT N.267
    TEXT268 : BOOL ;	//TEXT N.268
    TEXT269 : BOOL ;	//TEXT N.269
    TEXT270 : BOOL ;	//TEXT N.270
    TEXT271 : BOOL ;	//TEXT N.271
    TEXT272 : BOOL ;	//TEXT N.272
    TEXT257 : BOOL ;	//TEXT N.257
    TEXT258 : BOOL ;	//TEXT N.258
    TEXT259 : BOOL ;	//TEXT N.259
    TEXT260 : BOOL ;	//TEXT N.260
    TEXT261 : BOOL ;	//TEXT N.261
    TEXT262 : BOOL ;	//TEXT N.262
    TEXT263 : BOOL ;	//TEXT N.263
    TEXT264 : BOOL ;	//TEXT N.264
    TEXT281 : BOOL ;	//TEXT N.281
    TEXT282 : BOOL ;	//TEXT N.282
    TEXT283 : BOOL ;	//TEXT N.283
    TEXT284 : BOOL ;	//TEXT N.284
    TEXT285 : BOOL ;	//TEXT N.285
    TEXT286 : BOOL ;	//TEXT N.286
    TEXT287 : BOOL ;	//TEXT N.287
    TEXT288 : BOOL ;	//TEXT N.288
    TEXT273 : BOOL ;	//TEXT N.273
    TEXT274 : BOOL ;	//TEXT N.274
    TEXT275 : BOOL ;	//TEXT N.275
    TEXT276 : BOOL ;	//TEXT N.276
    TEXT277 : BOOL ;	//TEXT N.277
    TEXT278 : BOOL ;	//TEXT N.278
    TEXT279 : BOOL ;	//TEXT N.279
    TEXT280 : BOOL ;	//TEXT N.280
    TEXT297 : BOOL ;	//TEXT N.297
    TEXT298 : BOOL ;	//TEXT N.298
    TEXT299 : BOOL ;	//TEXT N.299
    TEXT300 : BOOL ;	//TEXT N.300
    TEXT301 : BOOL ;	//TEXT N.301
    TEXT302 : BOOL ;	//TEXT N.302
    TEXT303 : BOOL ;	//TEXT N.303
    TEXT304 : BOOL ;	//TEXT N.304
    TEXT289 : BOOL ;	//TEXT N.289
    TEXT290 : BOOL ;	//TEXT N.290
    TEXT291 : BOOL ;	//TEXT N.291
    TEXT292 : BOOL ;	//TEXT N.292
    TEXT293 : BOOL ;	//TEXT N.293
    TEXT294 : BOOL ;	//TEXT N.294
    TEXT295 : BOOL ;	//TEXT N.295
    TEXT296 : BOOL ;	//TEXT N.296
    TEXT313 : BOOL ;	//TEXT N.313
    TEXT314 : BOOL ;	//TEXT N.314
    TEXT315 : BOOL ;	//TEXT N.315
    TEXT316 : BOOL ;	//TEXT N.316
    TEXT317 : BOOL ;	//TEXT N.317
    TEXT318 : BOOL ;	//TEXT N.318
    TEXT319 : BOOL ;	//TEXT N.319
    TEXT320 : BOOL ;	//TEXT N.320
    TEXT305 : BOOL ;	//TEXT N.305
    TEXT306 : BOOL ;	//TEXT N.306
    TEXT307 : BOOL ;	//TEXT N.307
    TEXT308 : BOOL ;	//TEXT N.308
    TEXT309 : BOOL ;	//TEXT N.309
    TEXT310 : BOOL ;	//TEXT N.310
    TEXT311 : BOOL ;	//TEXT N.311
    TEXT312 : BOOL ;	//TEXT N.312
    TEXT329 : BOOL ;	//TEXT N.329
    TEXT330 : BOOL ;	//TEXT N.330
    TEXT331 : BOOL ;	//TEXT N.331
    TEXT332 : BOOL ;	//TEXT N.332
    TEXT333 : BOOL ;	//TEXT N.333
    TEXT334 : BOOL ;	//TEXT N.334
    TEXT335 : BOOL ;	//TEXT N.335
    TEXT336 : BOOL ;	//TEXT N.336
    TEXT321 : BOOL ;	//TEXT N.321
    TEXT322 : BOOL ;	//TEXT N.322
    TEXT323 : BOOL ;	//TEXT N.323
    TEXT324 : BOOL ;	//TEXT N.324
    TEXT325 : BOOL ;	//TEXT N.325
    TEXT326 : BOOL ;	//TEXT N.326
    TEXT327 : BOOL ;	//TEXT N.327
    TEXT328 : BOOL ;	//TEXT N.328
    TEXT345 : BOOL ;	//TEXT N.345
    TEXT346 : BOOL ;	//TEXT N.346
    TEXT347 : BOOL ;	//TEXT N.347
    TEXT348 : BOOL ;	//TEXT N.348
    TEXT349 : BOOL ;	//TEXT N.349
    TEXT350 : BOOL ;	//TEXT N.350
    TEXT351 : BOOL ;	//TEXT N.351
    TEXT352 : BOOL ;	//TEXT N.352
    TEXT337 : BOOL ;	//TEXT N.337
    TEXT338 : BOOL ;	//TEXT N.338
    TEXT339 : BOOL ;	//TEXT N.339
    TEXT340 : BOOL ;	//TEXT N.340
    TEXT341 : BOOL ;	//TEXT N.341
    TEXT342 : BOOL ;	//TEXT N.342
    TEXT343 : BOOL ;	//TEXT N.343
    TEXT344 : BOOL ;	//TEXT N.344
    TEXT361 : BOOL ;	//TEXT N.361
    TEXT362 : BOOL ;	//TEXT N.362
    TEXT363 : BOOL ;	//TEXT N.363
    TEXT364 : BOOL ;	//TEXT N.364
    TEXT365 : BOOL ;	//TEXT N.365
    TEXT366 : BOOL ;	//TEXT N.366
    TEXT367 : BOOL ;	//TEXT N.367
    TEXT368 : BOOL ;	//TEXT N.368
    TEXT353 : BOOL ;	//TEXT N.353
    TEXT354 : BOOL ;	//TEXT N.354
    TEXT355 : BOOL ;	//TEXT N.355
    TEXT356 : BOOL ;	//TEXT N.356
    TEXT357 : BOOL ;	//TEXT N.357
    TEXT358 : BOOL ;	//TEXT N.358
    TEXT359 : BOOL ;	//TEXT N.359
    TEXT360 : BOOL ;	//TEXT N.360
    TEXT377 : BOOL ;	//TEXT N.377
    TEXT378 : BOOL ;	//TEXT N.378
    TEXT379 : BOOL ;	//TEXT N.379
    TEXT380 : BOOL ;	//TEXT N.380
    TEXT381 : BOOL ;	//TEXT N.381
    TEXT382 : BOOL ;	//TEXT N.382
    TEXT383 : BOOL ;	//TEXT N.383
    TEXT384 : BOOL ;	//TEXT N.384
    TEXT369 : BOOL ;	//TEXT N.369
    TEXT370 : BOOL ;	//TEXT N.370
    TEXT371 : BOOL ;	//TEXT N.371
    TEXT372 : BOOL ;	//TEXT N.372
    TEXT373 : BOOL ;	//TEXT N.373
    TEXT374 : BOOL ;	//TEXT N.374
    TEXT375 : BOOL ;	//TEXT N.375
    TEXT376 : BOOL ;	//TEXT N.376
    TEXT393 : BOOL ;	//TEXT N.393
    TEXT394 : BOOL ;	//TEXT N.394
    TEXT395 : BOOL ;	//TEXT N.395
    TEXT396 : BOOL ;	//TEXT N.396
    TEXT397 : BOOL ;	//TEXT N.397
    TEXT398 : BOOL ;	//TEXT N.398
    TEXT399 : BOOL ;	//TEXT N.399
    TEXT400 : BOOL ;	//TEXT N.400
    TEXT385 : BOOL ;	//TEXT N.385
    TEXT386 : BOOL ;	//TEXT N.386
    TEXT387 : BOOL ;	//TEXT N.387
    TEXT388 : BOOL ;	//TEXT N.388
    TEXT389 : BOOL ;	//TEXT N.389
    TEXT390 : BOOL ;	//TEXT N.390
    TEXT391 : BOOL ;	//TEXT N.391
    TEXT392 : BOOL ;	//TEXT N.392
    TEXT409 : BOOL ;	//TEXT N.409
    TEXT410 : BOOL ;	//TEXT N.410
    TEXT411 : BOOL ;	//TEXT N.411
    TEXT412 : BOOL ;	//TEXT N.412
    TEXT413 : BOOL ;	//TEXT N.413
    TEXT414 : BOOL ;	//TEXT N.414
    TEXT415 : BOOL ;	//TEXT N.415
    TEXT416 : BOOL ;	//TEXT N.416
    TEXT401 : BOOL ;	//TEXT N.401
    TEXT402 : BOOL ;	//TEXT N.402
    TEXT403 : BOOL ;	//TEXT N.403
    TEXT404 : BOOL ;	//TEXT N.404
    TEXT405 : BOOL ;	//TEXT N.405
    TEXT406 : BOOL ;	//TEXT N.406
    TEXT407 : BOOL ;	//TEXT N.407
    TEXT408 : BOOL ;	//TEXT N.408
    TEXT425 : BOOL ;	//TEXT N.425
    TEXT426 : BOOL ;	//TEXT N.426
    TEXT427 : BOOL ;	//TEXT N.427
    TEXT428 : BOOL ;	//TEXT N.428
    TEXT429 : BOOL ;	//TEXT N.429
    TEXT430 : BOOL ;	//TEXT N.430
    TEXT431 : BOOL ;	//TEXT N.431
    TEXT432 : BOOL ;	//TEXT N.432
    TEXT417 : BOOL ;	//TEXT N.417
    TEXT418 : BOOL ;	//TEXT N.418
    TEXT419 : BOOL ;	//TEXT N.419
    TEXT420 : BOOL ;	//TEXT N.420
    TEXT421 : BOOL ;	//TEXT N.421
    TEXT422 : BOOL ;	//TEXT N.422
    TEXT423 : BOOL ;	//TEXT N.423
    TEXT424 : BOOL ;	//TEXT N.424
    TEXT441 : BOOL ;	//TEXT N.441
    TEXT442 : BOOL ;	//TEXT N.442
    TEXT443 : BOOL ;	//TEXT N.443
    TEXT444 : BOOL ;	//TEXT N.444
    TEXT445 : BOOL ;	//TEXT N.445
    TEXT446 : BOOL ;	//TEXT N.446
    TEXT447 : BOOL ;	//TEXT N.447
    TEXT448 : BOOL ;	//TEXT N.448
    TEXT433 : BOOL ;	//TEXT N.433
    TEXT434 : BOOL ;	//TEXT N.434
    TEXT435 : BOOL ;	//TEXT N.435
    TEXT436 : BOOL ;	//TEXT N.436
    TEXT437 : BOOL ;	//TEXT N.437
    TEXT438 : BOOL ;	//TEXT N.438
    TEXT439 : BOOL ;	//TEXT N.439
    TEXT440 : BOOL ;	//TEXT N.440
    TEXT457 : BOOL ;	//TEXT N.457
    TEXT458 : BOOL ;	//TEXT N.458
    TEXT459 : BOOL ;	//TEXT N.459
    TEXT460 : BOOL ;	//TEXT N.460
    TEXT461 : BOOL ;	//TEXT N.461
    TEXT462 : BOOL ;	//TEXT N.462
    TEXT463 : BOOL ;	//TEXT N.463
    TEXT464 : BOOL ;	//TEXT N.464
    TEXT449 : BOOL ;	//TEXT N.449
    TEXT450 : BOOL ;	//TEXT N.450
    TEXT451 : BOOL ;	//TEXT N.451
    TEXT452 : BOOL ;	//TEXT N.452
    TEXT453 : BOOL ;	//TEXT N.453
    TEXT454 : BOOL ;	//TEXT N.454
    TEXT455 : BOOL ;	//TEXT N.455
    TEXT456 : BOOL ;	//TEXT N.456
    TEXT473 : BOOL ;	//TEXT N.473
    TEXT474 : BOOL ;	//TEXT N.474
    TEXT475 : BOOL ;	//TEXT N.475
    TEXT476 : BOOL ;	//TEXT N.476
    TEXT477 : BOOL ;	//TEXT N.477
    TEXT478 : BOOL ;	//TEXT N.478
    TEXT479 : BOOL ;	//TEXT N.479
    TEXT480 : BOOL ;	//TEXT N.480
    TEXT465 : BOOL ;	//TEXT N.465
    TEXT466 : BOOL ;	//TEXT N.466
    TEXT467 : BOOL ;	//TEXT N.467
    TEXT468 : BOOL ;	//TEXT N.468
    TEXT469 : BOOL ;	//TEXT N.469
    TEXT470 : BOOL ;	//TEXT N.470
    TEXT471 : BOOL ;	//TEXT N.471
    TEXT472 : BOOL ;	//TEXT N.472
    TEXT489 : BOOL ;	//TEXT N.489
    TEXT490 : BOOL ;	//TEXT N.490
    TEXT491 : BOOL ;	//TEXT N.491
    TEXT492 : BOOL ;	//TEXT N.492
    TEXT493 : BOOL ;	//TEXT N.493
    TEXT494 : BOOL ;	//TEXT N.494
    TEXT495 : BOOL ;	//TEXT N.495
    TEXT496 : BOOL ;	//TEXT N.496
    TEXT481 : BOOL ;	//TEXT N.481
    TEXT482 : BOOL ;	//TEXT N.482
    TEXT483 : BOOL ;	//TEXT N.483
    TEXT484 : BOOL ;	//TEXT N.484
    TEXT485 : BOOL ;	//TEXT N.485
    TEXT486 : BOOL ;	//TEXT N.486
    TEXT487 : BOOL ;	//TEXT N.487
    TEXT488 : BOOL ;	//TEXT N.488
    TEXT505 : BOOL ;	//TEXT N.505
    TEXT506 : BOOL ;	//TEXT N.506
    TEXT507 : BOOL ;	//TEXT N.507
    TEXT508 : BOOL ;	//TEXT N.508
    TEXT509 : BOOL ;	//TEXT N.509
    TEXT510 : BOOL ;	//TEXT N.510
    TEXT511 : BOOL ;	//TEXT N.511
    TEXT512 : BOOL ;	//TEXT N.512
    TEXT497 : BOOL ;	//TEXT N.497
    TEXT498 : BOOL ;	//TEXT N.498
    TEXT499 : BOOL ;	//TEXT N.499
    TEXT500 : BOOL ;	//TEXT N.500
    TEXT501 : BOOL ;	//TEXT N.501
    TEXT502 : BOOL ;	//TEXT N.502
    TEXT503 : BOOL ;	//TEXT N.503
    TEXT504 : BOOL ;	//TEXT N.504
    TEXT521 : BOOL ;	//TEXT N.521
    TEXT522 : BOOL ;	//TEXT N.522
    TEXT523 : BOOL ;	//TEXT N.523
    TEXT524 : BOOL ;	//TEXT N.524
    TEXT525 : BOOL ;	//TEXT N.525
    TEXT526 : BOOL ;	//TEXT N.526
    TEXT527 : BOOL ;	//TEXT N.527
    TEXT528 : BOOL ;	//TEXT N.528
    TEXT513 : BOOL ;	//TEXT N.513
    TEXT514 : BOOL ;	//TEXT N.514
    TEXT515 : BOOL ;	//TEXT N.515
    TEXT516 : BOOL ;	//TEXT N.516
    TEXT517 : BOOL ;	//TEXT N.517
    TEXT518 : BOOL ;	//TEXT N.518
    TEXT519 : BOOL ;	//TEXT N.519
    TEXT520 : BOOL ;	//TEXT N.520
    TEXT537 : BOOL ;	//TEXT N.537
    TEXT538 : BOOL ;	//TEXT N.538
    TEXT539 : BOOL ;	//TEXT N.539
    TEXT540 : BOOL ;	//TEXT N.540
    TEXT541 : BOOL ;	//TEXT N.541
    TEXT542 : BOOL ;	//TEXT N.542
    TEXT543 : BOOL ;	//TEXT N.543
    TEXT544 : BOOL ;	//TEXT N.544
    TEXT529 : BOOL ;	//TEXT N.529
    TEXT530 : BOOL ;	//TEXT N.530
    TEXT531 : BOOL ;	//TEXT N.531
    TEXT532 : BOOL ;	//TEXT N.532
    TEXT533 : BOOL ;	//TEXT N.533
    TEXT534 : BOOL ;	//TEXT N.534
    TEXT535 : BOOL ;	//TEXT N.535
    TEXT536 : BOOL ;	//TEXT N.536
    TEXT553 : BOOL ;	//TEXT N.553
    TEXT554 : BOOL ;	//TEXT N.554
    TEXT555 : BOOL ;	//TEXT N.555
    TEXT556 : BOOL ;	//TEXT N.556
    TEXT557 : BOOL ;	//TEXT N.557
    TEXT558 : BOOL ;	//TEXT N.558
    TEXT559 : BOOL ;	//TEXT N.559
    TEXT560 : BOOL ;	//TEXT N.560
    TEXT545 : BOOL ;	//TEXT N.545
    TEXT546 : BOOL ;	//TEXT N.546
    TEXT547 : BOOL ;	//TEXT N.547
    TEXT548 : BOOL ;	//TEXT N.548
